KUKA KRL program: EPS_2_251806_MH13A_A_20260223023042.src

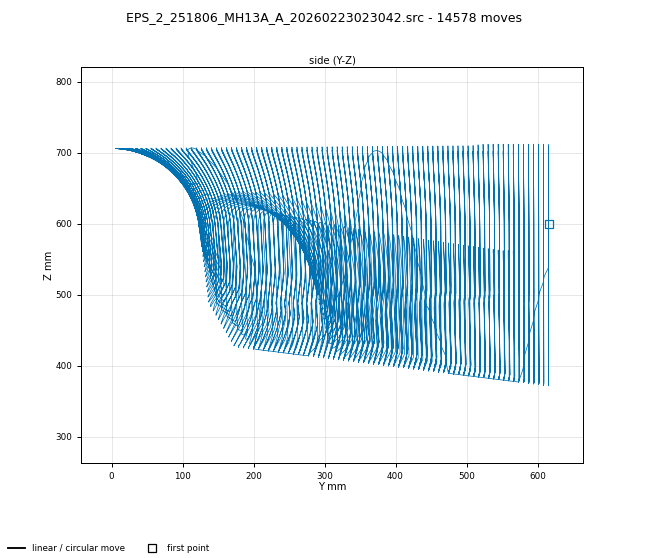
[picture p0: tool path of EPS_2_251806_MH13A_A_20260223023042.src, 14578 of 14580 moves have a stored position in this frame; points joined in program order, loops and branches not executed]
&ACCESS RVP
&REL 4
&COMMENT QRS 19112012
&PARAM EDITMASK = *
DEF PART()
EXT BAS (BAS_COMMAND :IN,REAL :IN )
INT I
BAS (#INITMOV,0 )

;KUKA QRS Post kuka4.cps  Date:22-06-2017 !

File_ID=3082

QRS_PRE_INIT()

;Init var - Until changes are made in qrs_pre_init
Outlet_Square_prg=0
Inlet_1_Square_prg=0
Inlet_2_Square_prg=0
Inlet_3_Square_prg=0
Inlet_4_Square_prg=0
Inlet_5_Square_prg=0

Outlet_1={X 0.000, Y 524.580, Z 611.500, B 0.000, E1 0.000 }
Inlet_1={X 0.000, Y 548.820, Z 271.500, B 0.000, E1 90.000 }
Inlet_2={X 0.000, Y 525.290, Z 601.500, B 0.000, E1 180.000 }
Outlet_1_type=201
Inlet_1_type=201
Inlet_2_type=201
;QRS#1=Sidecore dimensions
;QRS#2=200-8" PVC SDR 35
;QRS#3=200-8" PVC SDR 35
;QRS#4=200-8" PVC SDR 35
;QRS#5=
;QRS#6=
;QRS#7=
;QRS#8=
;QRS#9=12-08 PSX
;QRS#10=12-08 PSX
;QRS#11=12-08 PSX
;QRS#12=
;QRS#13=
;QRS#14=
;QRS#15=
;QRS#16=1220x127x991 3,25'
;QRS#17=EPS Height
;QRS#18=712
;QRS#19=*
;QRS#20= UPDATED VERSION 22-06-2017
;QRS#21=*
Outlet_Square=0100
Inlet_1_Square=0100
Inlet_2_Square=0100
Inlet_3_Square=0
Inlet_4_Square=0
Inlet_5_Square=0
Mill_Square=1
Outlet_Square_Prg=204
Inlet_1_Square_prg=204
Inlet_2_Square_prg=204

QRS_INIT()

$ADVANCE=5

; T1
PTP {E1 173.498,E2 173.498}
PTP {X 0,Y 615.498,A -85,B 0,C 180,E1 173.498,E2 173.498,E3 0,E4 0,E5 0,E6 0}
QRS_SPEED_INIT()
LIN {X 0,Y 615.498,Z 600,A -85,B 0,C 180,E1 173.498,E2 173.498,E3 0,E4 0,E5 0,E6 0} C_VEL
LIN {X 0,Y 615.498,Z 552.731,A -85,B 0,C 180,E1 173.498,E2 173.498} C_VEL
LIN {X 0,Y 615.498,Z 541.852,A -85,B 0,C 180,E1 173.498,E2 173.498} C_VEL
LIN {X 0,Y 615.496,Z 540.208,A -85,B 0,C 180,E1 173.418,E2 173.418} C_VEL
LIN {X 0,Y 615.497,Z 532.536,A -85,B 0,C 180,E1 172.455,E2 172.455} C_VEL
LIN {X 0,Y 615.498,Z 522.758,A -85,B 0,C 180,E1 171.463,E2 171.463} C_VEL
LIN {X 0,Y 615.498,Z 512.492,A -85,B 0,C 180,E1 170.636,E2 170.636} C_VEL
LIN {X 0,Y 615.496,Z 500.928,A -85,B 0,C 180,E1 169.889,E2 169.889} C_VEL
LIN {X 0,Y 615.499,Z 489.021,A -85,B 0,C 180,E1 169.291,E2 169.291} C_VEL
LIN {X 0,Y 615.498,Z 476.155,A -85,B 0,C 180,E1 168.807,E2 168.807} C_VEL
LIN {X 0,Y 615.497,Z 463.553,A -85,B 0,C 180,E1 168.473,E2 168.473} C_VEL
LIN {X 0,Y 615.498,Z 450.425,A -85,B 0,C 180,E1 168.265,E2 168.265} C_VEL
LIN {X 0,Y 615.498,Z 372.93,A -85,B 0,C 180,E1 167.344,E2 167.344} C_VEL
LIN {X 0,Y 615.495,Z 371.855,A -85,B 0,C 180,E1 167.218,E2 167.218} C_VEL
LIN {X 0,Y 615.472,Z 371.694,A -85,B 0,C 180,E1 164.773,E2 164.773} C_VEL
LIN {X 0,Y 615.491,Z 371.682,A -85,B 0,C 180,E1 162.043,E2 162.043} C_VEL
LIN {X 0,Y 615.495,Z 371.698,A -85,B 0,C 180,E1 159.269,E2 159.269} C_VEL
LIN {X 0,Y 615.469,Z 371.687,A -85,B 0,C 180,E1 156.443,E2 156.443} C_VEL
LIN {X 0,Y 615.487,Z 371.692,A -85,B 0,C 180,E1 153.556,E2 153.556} C_VEL
LIN {X 0,Y 615.491,Z 371.699,A -85,B 0,C 180,E1 151.342,E2 151.342} C_VEL
LIN {X 0,Y 615.47,Z 371.695,A -85,B 0,C 180,E1 148.917,E2 148.917} C_VEL
LIN {X 0,Y 615.464,Z 371.688,A -85,B 0,C 180,E1 146.47,E2 146.47} C_VEL
LIN {X 0,Y 615.483,Z 371.684,A -85,B 0,C 180,E1 144.167,E2 144.167} C_VEL
LIN {X 0,Y 615.475,Z 371.697,A -85,B 0,C 180,E1 141.094,E2 141.094} C_VEL
LIN {X 0,Y 615.46,Z 371.689,A -85,B 0,C 180,E1 138.524,E2 138.524} C_VEL
LIN {X 0,Y 615.493,Z 371.686,A -85,B 0,C 180,E1 135.851,E2 135.851} C_VEL
LIN {X 0,Y 615.467,Z 371.696,A -85,B 0,C 180,E1 133.045,E2 133.045} C_VEL
LIN {X 0,Y 615.455,Z 371.69,A -85,B 0,C 180,E1 130.609,E2 130.609} C_VEL
LIN {X 0,Y 615.482,Z 371.687,A -85,B 0,C 180,E1 128.011,E2 128.011} C_VEL
LIN {X 0,Y 615.494,Z 371.695,A -85,B 0,C 180,E1 125.616,E2 125.616} C_VEL
LIN {X 0,Y 615.474,Z 371.698,A -85,B 0,C 180,E1 123.237,E2 123.237} C_VEL
LIN {X 0,Y 615.452,Z 371.694,A -85,B 0,C 180,E1 120.922,E2 120.922} C_VEL
LIN {X 0,Y 615.457,Z 371.689,A -85,B 0,C 180,E1 118.444,E2 118.444} C_VEL
LIN {X 0,Y 615.494,Z 371.701,A -85,B 0,C 180,E1 115.569,E2 115.569} C_VEL
LIN {X 0,Y 615.498,Z 372.248,A -85,B 0,C 180,E1 115.334,E2 115.334} C_VEL
LIN {X 0,Y 615.455,Z 395.722,A -85,B 0,C 180,E1 112.721,E2 112.721} C_VEL
LIN {X 0,Y 615.489,Z 421.96,A -85,B 0,C 180,E1 109.859,E2 109.859} C_VEL
LIN {X 0,Y 615.449,Z 447.71,A -85,B 0,C 180,E1 107.1,E2 107.1} C_VEL
LIN {X 0,Y 615.495,Z 473.284,A -85,B 0,C 180,E1 104.395,E2 104.395} C_VEL
LIN {X 0,Y 615.494,Z 488.065,A -85,B 0,C 180,E1 102.865,E2 102.865} C_VEL
LIN {X 0,Y 615.482,Z 504.142,A -85,B 0,C 180,E1 102.656,E2 102.656} C_VEL
LIN {X 0,Y 615.493,Z 597.644,A -85,B 0,C 180,E1 101.547,E2 101.547} C_VEL
LIN {X 0,Y 615.499,Z 610.222,A -85,B 0,C 180,E1 101.276,E2 101.276} C_VEL
LIN {X 0,Y 615.497,Z 623.523,A -85,B 0,C 180,E1 100.845,E2 100.845} C_VEL
LIN {X 0,Y 615.493,Z 634.565,A -85,B 0,C 180,E1 100.36,E2 100.36} C_VEL
LIN {X 0,Y 615.491,Z 646.305,A -85,B 0,C 180,E1 99.696,E2 99.696} C_VEL
LIN {X 0,Y 615.499,Z 656.768,A -85,B 0,C 180,E1 98.95,E2 98.95} C_VEL
LIN {X 0,Y 615.498,Z 665.331,A -85,B 0,C 180,E1 98.206,E2 98.206} C_VEL
LIN {X 0,Y 615.497,Z 673.21,A -85,B 0,C 180,E1 97.38,E2 97.38} C_VEL
LIN {X 0,Y 615.497,Z 680.899,A -85,B 0,C 180,E1 96.392,E2 96.392} C_VEL
LIN {X 0,Y 615.497,Z 687.958,A -85,B 0,C 180,E1 95.241,E2 95.241} C_VEL
LIN {X 0,Y 615.494,Z 692.658,A -85,B 0,C 180,E1 94.256,E2 94.256} C_VEL
LIN {X 0,Y 615.494,Z 696.255,A -85,B 0,C 180,E1 93.273,E2 93.273} C_VEL
LIN {X 0,Y 615.496,Z 698.115,A -85,B 0,C 180,E1 92.618,E2 92.618} C_VEL
LIN {X 0,Y 615.499,Z 699.533,A -85,B 0,C 180,E1 91.963,E2 91.963} C_VEL
LIN {X 0,Y 615.496,Z 701.142,A -85,B 0,C 180,E1 90.654,E2 90.654} C_VEL
LIN {X 0,Y 615.495,Z 701.384,A -85,B 0,C 180,E1 90,E2 90} C_VEL
LIN {X 0,Y 615.495,Z 701.206,A -85,B 0,C 180,E1 89.346,E2 89.346} C_VEL
LIN {X 0,Y 615.499,Z 699.682,A -85,B 0,C 180,E1 88.037,E2 88.037} C_VEL
LIN {X 0,Y 615.498,Z 698.341,A -85,B 0,C 180,E1 87.382,E2 87.382} C_VEL
LIN {X 0,Y 615.496,Z 695.494,A -85,B 0,C 180,E1 86.399,E2 86.399} C_VEL
LIN {X 0,Y 615.498,Z 691.634,A -85,B 0,C 180,E1 85.415,E2 85.415} C_VEL
LIN {X 0,Y 615.498,Z 686.651,A -85,B 0,C 180,E1 84.43,E2 84.43} C_VEL
LIN {X 0,Y 615.496,Z 680.208,A -85,B 0,C 180,E1 83.418,E2 83.418} C_VEL
LIN {X 0,Y 615.497,Z 672.535,A -85,B 0,C 180,E1 82.454,E2 82.454} C_VEL
LIN {X 0,Y 615.498,Z 662.757,A -85,B 0,C 180,E1 81.463,E2 81.463} C_VEL
LIN {X 0,Y 615.498,Z 652.491,A -85,B 0,C 180,E1 80.635,E2 80.635} C_VEL
LIN {X 0,Y 615.492,Z 640.927,A -85,B 0,C 180,E1 79.889,E2 79.889} C_VEL
LIN {X 0,Y 615.497,Z 629.02,A -85,B 0,C 180,E1 79.291,E2 79.291} C_VEL
LIN {X 0,Y 615.498,Z 616.153,A -85,B 0,C 180,E1 78.807,E2 78.807} C_VEL
LIN {X 0,Y 615.493,Z 603.55,A -85,B 0,C 180,E1 78.473,E2 78.473} C_VEL
LIN {X 0,Y 615.491,Z 590.42,A -85,B 0,C 180,E1 78.264,E2 78.264} C_VEL
LIN {X 0,Y 615.489,Z 488.172,A -85,B 0,C 180,E1 77.05,E2 77.05} C_VEL
LIN {X 0,Y 615.453,Z 466.245,A -85,B 0,C 180,E1 74.773,E2 74.773} C_VEL
LIN {X 0,Y 615.495,Z 440.506,A -85,B 0,C 180,E1 72.043,E2 72.043} C_VEL
LIN {X 0,Y 615.494,Z 414.735,A -85,B 0,C 180,E1 69.269,E2 69.269} C_VEL
LIN {X 0,Y 615.448,Z 390.567,A -85,B 0,C 180,E1 66.62,E2 66.62} C_VEL
LIN {X 0,Y 615.497,Z 372.017,A -85,B 0,C 180,E1 64.539,E2 64.539} C_VEL
LIN {X 0,Y 615.497,Z 371.697,A -85,B 0,C 180,E1 64.284,E2 64.284} C_VEL
LIN {X 0,Y 615.441,Z 371.692,A -85,B 0,C 180,E1 61.339,E2 61.339} C_VEL
LIN {X 0,Y 615.445,Z 371.696,A -85,B 0,C 180,E1 58.921,E2 58.921} C_VEL
LIN {X 0,Y 615.492,Z 371.689,A -85,B 0,C 180,E1 55.978,E2 55.978} C_VEL
LIN {X 0,Y 615.451,Z 371.691,A -85,B 0,C 180,E1 53.572,E2 53.572} C_VEL
LIN {X 0,Y 615.442,Z 371.696,A -85,B 0,C 180,E1 50.944,E2 50.944} C_VEL
LIN {X 0,Y 615.471,Z 371.7,A -85,B 0,C 180,E1 48.524,E2 48.524} C_VEL
LIN {X 0,Y 615.479,Z 371.689,A -85,B 0,C 180,E1 45.849,E2 45.849} C_VEL
LIN {X 0,Y 615.436,Z 371.693,A -85,B 0,C 180,E1 43.249,E2 43.249} C_VEL
LIN {X 0,Y 615.436,Z 371.695,A -85,B 0,C 180,E1 41.088,E2 41.088} C_VEL
LIN {X 0,Y 615.441,Z 371.696,A -85,B 0,C 180,E1 38.908,E2 38.908} C_VEL
LIN {X 0,Y 615.479,Z 371.701,A -85,B 0,C 180,E1 36.426,E2 36.426} C_VEL
LIN {X 0,Y 615.447,Z 371.692,A -85,B 0,C 180,E1 33.528,E2 33.528} C_VEL
LIN {X 0,Y 615.434,Z 371.695,A -85,B 0,C 180,E1 31.077,E2 31.077} C_VEL
LIN {X 0,Y 615.479,Z 371.699,A -85,B 0,C 180,E1 28.448,E2 28.448} C_VEL
LIN {X 0,Y 615.448,Z 371.692,A -85,B 0,C 180,E1 25.56,E2 25.56} C_VEL
LIN {X 0,Y 615.448,Z 371.692,A -85,B 0,C 180,E1 23.558,E2 23.558} C_VEL
LIN {X 0,Y 615.439,Z 371.693,A -85,B 0,C 180,E1 21.434,E2 21.434} C_VEL
LIN {X 0,Y 615.435,Z 371.694,A -85,B 0,C 180,E1 19.34,E2 19.34} C_VEL
LIN {X 0,Y 615.431,Z 371.694,A -85,B 0,C 180,E1 17.272,E2 17.272} C_VEL
LIN {X 0,Y 615.431,Z 371.695,A -85,B 0,C 180,E1 15.228,E2 15.228} C_VEL
LIN {X 0,Y 615.43,Z 371.695,A -85,B 0,C 180,E1 13.203,E2 13.203} C_VEL
LIN {X 0,Y 615.436,Z 371.697,A -85,B 0,C 180,E1 10.861,E2 10.861} C_VEL
LIN {X 0,Y 615.461,Z 371.698,A -85,B 0,C 180,E1 8.537,E2 8.537} C_VEL
LIN {X 0,Y 615.484,Z 371.692,A -85,B 0,C 180,E1 5.899,E2 5.899} C_VEL
LIN {X 0,Y 615.43,Z 371.695,A -85,B 0,C 180,E1 3.273,E2 3.273} C_VEL
LIN {X 0,Y 615.431,Z 371.695,A -85,B 0,C 180,E1 1.309,E2 1.309} C_VEL
LIN {X 0,Y 615.432,Z 371.695,A -85,B 0,C 180,E1 -0.654,E2 -0.654} C_VEL
LIN {X 0,Y 615.433,Z 371.694,A -85,B 0,C 180,E1 -2.618,E2 -2.618} C_VEL
LIN {X 0,Y 615.435,Z 371.694,A -85,B 0,C 180,E1 -4.585,E2 -4.585} C_VEL
LIN {X 0,Y 615.436,Z 371.694,A -85,B 0,C 180,E1 -6.557,E2 -6.557} C_VEL
LIN {X 0,Y 615.437,Z 371.694,A -85,B 0,C 180,E1 -8.537,E2 -8.537} C_VEL
LIN {X 0,Y 615.425,Z 371.696,A -85,B 0,C 180,E1 -10.855,E2 -10.855} C_VEL
LIN {X 0,Y 615.433,Z 371.697,A -85,B 0,C 180,E1 -13.202,E2 -13.202} C_VEL
LIN {X 0,Y 615.49,Z 371.699,A -85,B 0,C 180,E1 -15.905,E2 -15.905} C_VEL
LIN {X 0,Y 615.429,Z 371.696,A -85,B 0,C 180,E1 -18.648,E2 -18.648} C_VEL
LIN {X 0,Y 615.426,Z 371.696,A -85,B 0,C 180,E1 -20.733,E2 -20.733} C_VEL
LIN {X 0,Y 615.423,Z 371.696,A -85,B 0,C 180,E1 -22.847,E2 -22.847} C_VEL
LIN {X 0,Y 615.423,Z 371.697,A -85,B 0,C 180,E1 -24.995,E2 -24.995} C_VEL
LIN {X 0,Y 615.483,Z 371.701,A -85,B 0,C 180,E1 -27.915,E2 -27.915} C_VEL
LIN {X 0,Y 615.475,Z 371.694,A -85,B 0,C 180,E1 -30.161,E2 -30.161} C_VEL
LIN {X 0,Y 615.441,Z 371.695,A -85,B 0,C 180,E1 -32.46,E2 -32.46} C_VEL
LIN {X 0,Y 615.421,Z 371.697,A -85,B 0,C 180,E1 -34.819,E2 -34.819} C_VEL
LIN {X 0,Y 615.429,Z 371.698,A -85,B 0,C 180,E1 -37.246,E2 -37.246} C_VEL
LIN {X 0,Y 615.486,Z 371.695,A -85,B 0,C 180,E1 -40.088,E2 -40.088} C_VEL
LIN {X 0,Y 615.45,Z 371.696,A -85,B 0,C 180,E1 -42.356,E2 -42.356} C_VEL
LIN {X 0,Y 615.417,Z 371.698,A -85,B 0,C 180,E1 -44.924,E2 -44.924} C_VEL
LIN {X 0,Y 615.417,Z 371.698,A -85,B 0,C 180,E1 -46.96,E2 -46.96} C_VEL
LIN {X 0,Y 615.417,Z 371.698,A -85,B 0,C 180,E1 -48.913,E2 -48.913} C_VEL
LIN {X 0,Y 615.419,Z 371.698,A -85,B 0,C 180,E1 -51.09,E2 -51.09} C_VEL
LIN {X 0,Y 615.453,Z 371.699,A -85,B 0,C 180,E1 -53.572,E2 -53.572} C_VEL
LIN {X 0,Y 615.437,Z 371.697,A -85,B 0,C 180,E1 -56.473,E2 -56.473} C_VEL
LIN {X 0,Y 615.415,Z 371.699,A -85,B 0,C 180,E1 -59.076,E2 -59.076} C_VEL
LIN {X 0,Y 615.448,Z 371.699,A -85,B 0,C 180,E1 -61.557,E2 -61.557} C_VEL
LIN {X 0,Y 615.498,Z 371.811,A -85,B 0,C 180,E1 -64.012,E2 -64.012} C_VEL
LIN {X 0,Y 615.497,Z 372.154,A -85,B 0,C 180,E1 -64.103,E2 -64.103} C_VEL
LIN {X 0,Y 615.463,Z 395.618,A -85,B 0,C 180,E1 -66.621,E2 -66.621} C_VEL
LIN {X 0,Y 615.473,Z 420.833,A -85,B 0,C 180,E1 -69.269,E2 -69.269} C_VEL
LIN {X 0,Y 615.496,Z 447.725,A -85,B 0,C 180,E1 -72.043,E2 -72.043} C_VEL
LIN {X 0,Y 615.456,Z 474.585,A -85,B 0,C 180,E1 -74.773,E2 -74.773} C_VEL
LIN {X 0,Y 615.491,Z 497.862,A -85,B 0,C 180,E1 -77.092,E2 -77.092} C_VEL
LIN {X 0,Y 615.492,Z 607.82,A -85,B 0,C 180,E1 -78.411,E2 -78.411} C_VEL
LIN {X 0,Y 615.499,Z 620.336,A -85,B 0,C 180,E1 -78.682,E2 -78.682} C_VEL
LIN {X 0,Y 615.496,Z 633.5,A -85,B 0,C 180,E1 -79.109,E2 -79.109} C_VEL
LIN {X 0,Y 615.491,Z 645.473,A -85,B 0,C 180,E1 -79.639,E2 -79.639} C_VEL
LIN {X 0,Y 615.492,Z 656.992,A -85,B 0,C 180,E1 -80.304,E2 -80.304} C_VEL
LIN {X 0,Y 615.499,Z 667.339,A -85,B 0,C 180,E1 -81.05,E2 -81.05} C_VEL
LIN {X 0,Y 615.497,Z 675.81,A -85,B 0,C 180,E1 -81.794,E2 -81.794} C_VEL
LIN {X 0,Y 615.498,Z 683.605,A -85,B 0,C 180,E1 -82.619,E2 -82.619} C_VEL
LIN {X 0,Y 615.496,Z 691.202,A -85,B 0,C 180,E1 -83.608,E2 -83.608} C_VEL
LIN {X 0,Y 615.498,Z 698.204,A -85,B 0,C 180,E1 -84.759,E2 -84.759} C_VEL
LIN {X 0,Y 615.494,Z 702.851,A -85,B 0,C 180,E1 -85.743,E2 -85.743} C_VEL
LIN {X 0,Y 615.494,Z 706.398,A -85,B 0,C 180,E1 -86.727,E2 -86.727} C_VEL
LIN {X 0,Y 615.497,Z 708.233,A -85,B 0,C 180,E1 -87.382,E2 -87.382} C_VEL
LIN {X 0,Y 615.499,Z 709.607,A -85,B 0,C 180,E1 -88.037,E2 -88.037} C_VEL
LIN {X 0,Y 615.496,Z 711.173,A -85,B 0,C 180,E1 -89.346,E2 -89.346} C_VEL
LIN {X 0,Y 615.494,Z 711.389,A -85,B 0,C 180,E1 -90,E2 -90} C_VEL
LIN {X 0,Y 615.495,Z 710.58,A -85,B 0,C 180,E1 -91.308,E2 -91.308} C_VEL
LIN {X 0,Y 615.499,Z 709.608,A -85,B 0,C 180,E1 -91.963,E2 -91.963} C_VEL
LIN {X 0,Y 615.497,Z 708.233,A -85,B 0,C 180,E1 -92.618,E2 -92.618} C_VEL
LIN {X 0,Y 615.496,Z 705.35,A -85,B 0,C 180,E1 -93.601,E2 -93.601} C_VEL
LIN {X 0,Y 615.498,Z 701.442,A -85,B 0,C 180,E1 -94.584,E2 -94.584} C_VEL
LIN {X 0,Y 615.499,Z 696.405,A -85,B 0,C 180,E1 -95.57,E2 -95.57} C_VEL
LIN {X 0,Y 615.497,Z 689.869,A -85,B 0,C 180,E1 -96.583,E2 -96.583} C_VEL
LIN {X 0,Y 615.497,Z 682.133,A -85,B 0,C 180,E1 -97.545,E2 -97.545} C_VEL
LIN {X 0,Y 615.498,Z 674.045,A -85,B 0,C 180,E1 -98.371,E2 -98.371} C_VEL
LIN {X 0,Y 615.499,Z 664.168,A -85,B 0,C 180,E1 -99.199,E2 -99.199} C_VEL
LIN {X 0,Y 615.492,Z 652.981,A -85,B 0,C 180,E1 -99.945,E2 -99.945} C_VEL
LIN {X 0,Y 615.493,Z 642.022,A -85,B 0,C 180,E1 -100.527,E2 -100.527} C_VEL
LIN {X 0,Y 615.499,Z 629.416,A -85,B 0,C 180,E1 -101.042,E2 -101.042} C_VEL
LIN {X 0,Y 615.498,Z 617.063,A -85,B 0,C 180,E1 -101.401,E2 -101.401} C_VEL
LIN {X 0,Y 615.491,Z 603.466,A -85,B 0,C 180,E1 -101.652,E2 -101.652} C_VEL
LIN {X 0,Y 615.491,Z 497.865,A -85,B 0,C 180,E1 -102.907,E2 -102.907} C_VEL
LIN {X 0,Y 615.456,Z 474.586,A -85,B 0,C 180,E1 -105.227,E2 -105.227} C_VEL
LIN {X 0,Y 615.496,Z 447.727,A -85,B 0,C 180,E1 -107.957,E2 -107.957} C_VEL
LIN {X 0,Y 615.473,Z 420.835,A -85,B 0,C 180,E1 -110.731,E2 -110.731} C_VEL
LIN {X 0,Y 615.463,Z 395.62,A -85,B 0,C 180,E1 -113.379,E2 -113.379} C_VEL
LIN {X 0,Y 615.495,Z 372.155,A -85,B 0,C 180,E1 -115.897,E2 -115.897} C_VEL
LIN {X 0,Y 615.496,Z 371.721,A -85,B 0,C 180,E1 -116.079,E2 -116.079} C_VEL
LIN {X 0,Y 615.423,Z 371.7,A -85,B 0,C 180,E1 -118.661,E2 -118.661} C_VEL
LIN {X 0,Y 615.411,Z 371.7,A -85,B 0,C 180,E1 -121.074,E2 -121.074} C_VEL
LIN {X 0,Y 615.441,Z 371.7,A -85,B 0,C 180,E1 -123.527,E2 -123.527} C_VEL
LIN {X 0,Y 615.443,Z 371.697,A -85,B 0,C 180,E1 -126.428,E2 -126.428} C_VEL
LIN {X 0,Y 615.421,Z 371.698,A -85,B 0,C 180,E1 -128.91,E2 -128.91} C_VEL
LIN {X 0,Y 615.427,Z 371.698,A -85,B 0,C 180,E1 -131.088,E2 -131.088} C_VEL
LIN {X 0,Y 615.438,Z 371.698,A -85,B 0,C 180,E1 -133.249,E2 -133.249} C_VEL
LIN {X 0,Y 615.486,Z 371.694,A -85,B 0,C 180,E1 -136.003,E2 -136.003} C_VEL
LIN {X 0,Y 615.444,Z 371.693,A -85,B 0,C 180,E1 -138.522,E2 -138.522} C_VEL
LIN {X 0,Y 615.438,Z 371.695,A -85,B 0,C 180,E1 -140.944,E2 -140.944} C_VEL
LIN {X 0,Y 615.482,Z 371.702,A -85,B 0,C 180,E1 -143.575,E2 -143.575} C_VEL
LIN {X 0,Y 615.453,Z 371.691,A -85,B 0,C 180,E1 -146.471,E2 -146.471} C_VEL
LIN {X 0,Y 615.456,Z 371.696,A -85,B 0,C 180,E1 -149.078,E2 -149.078} C_VEL
LIN {X 0,Y 615.494,Z 371.699,A -85,B 0,C 180,E1 -151.549,E2 -151.549} C_VEL
LIN {X 0,Y 615.46,Z 371.689,A -85,B 0,C 180,E1 -154.437,E2 -154.437} C_VEL
LIN {X 0,Y 615.474,Z 371.698,A -85,B 0,C 180,E1 -157.155,E2 -157.155} C_VEL
LIN {X 0,Y 615.487,Z 371.686,A -85,B 0,C 180,E1 -159.967,E2 -159.967} C_VEL
LIN {X 0,Y 615.462,Z 371.692,A -85,B 0,C 180,E1 -162.729,E2 -162.729} C_VEL
LIN {X 0,Y 615.486,Z 371.696,A -85,B 0,C 180,E1 -165.451,E2 -165.451} C_VEL
LIN {X 0,Y 615.496,Z 371.905,A -85,B 0,C 180,E1 -167.323,E2 -167.323} C_VEL
LIN {X 0,Y 615.497,Z 372.808,A -85,B 0,C 180,E1 -167.428,E2 -167.428} C_VEL
LIN {X 0,Y 615.497,Z 458.789,A -85,B 0,C 180,E1 -168.473,E2 -168.473} C_VEL
LIN {X 0,Y 615.498,Z 471.737,A -85,B 0,C 180,E1 -168.765,E2 -168.765} C_VEL
LIN {X 0,Y 615.498,Z 484.736,A -85,B 0,C 180,E1 -169.2,E2 -169.2} C_VEL
LIN {X 0,Y 615.497,Z 496.194,A -85,B 0,C 180,E1 -169.723,E2 -169.723} C_VEL
LIN {X 0,Y 615.491,Z 507.576,A -85,B 0,C 180,E1 -170.387,E2 -170.387} C_VEL
LIN {X 0,Y 615.498,Z 517.823,A -85,B 0,C 180,E1 -171.133,E2 -171.133} C_VEL
LIN {X 0,Y 615.499,Z 527.034,A -85,B 0,C 180,E1 -171.959,E2 -171.959} C_VEL
LIN {X 0,Y 615.499,Z 535.892,A -85,B 0,C 180,E1 -172.943,E2 -172.943} C_VEL
LIN {X 0,Y 615.497,Z 543.123,A -85,B 0,C 180,E1 -173.937,E2 -173.937} C_VEL
LIN {X 0,Y 615.497,Z 547.958,A -85,B 0,C 180,E1 -174.759,E2 -174.759} C_VEL
LIN {X 0,Y 615.494,Z 552.658,A -85,B 0,C 180,E1 -175.744,E2 -175.744} C_VEL
LIN {X 0,Y 615.494,Z 556.255,A -85,B 0,C 180,E1 -176.727,E2 -176.727} C_VEL
LIN {X 0,Y 615.496,Z 558.115,A -85,B 0,C 180,E1 -177.382,E2 -177.382} C_VEL
LIN {X 0,Y 615.499,Z 559.533,A -85,B 0,C 180,E1 -178.037,E2 -178.037} C_VEL
LIN {X 0,Y 615.496,Z 561.142,A -85,B 0,C 180,E1 -179.346,E2 -179.346} C_VEL
LIN {X 0,Y 615.495,Z 561.384,A -85,B 0,C 180,E1 -180,E2 -180} C_VEL
LIN {X 0,Y 615.495,Z 561.206,A -85,B 0,C 180,E1 -180.654,E2 -180.654} C_VEL
LIN {X 0,Y 615.499,Z 559.682,A -85,B 0,C 180,E1 -181.963,E2 -181.963} C_VEL
LIN {X 0,Y 615.498,Z 558.341,A -85,B 0,C 180,E1 -182.618,E2 -182.618} C_VEL
LIN {X 0,Y 615.496,Z 555.494,A -85,B 0,C 180,E1 -183.601,E2 -183.601} C_VEL
LIN {X 0,Y 615.498,Z 551.634,A -85,B 0,C 180,E1 -184.585,E2 -184.585} C_VEL
LIN {X 0,Y 615.498,Z 546.651,A -85,B 0,C 180,E1 -185.57,E2 -185.57} C_VEL
LIN {X 0,Y 615.496,Z 540.208,A -85,B 0,C 180,E1 -186.582,E2 -186.582} C_VEL
LIN {X 0,Y 614.829,Z 537.026,A -85,B 0,C 180,E1 -187.031,E2 -187.031} C_VEL
LIN {X 0,Y 611.989,Z 531.453,A -85,B 0,C 180,E1 -187.748,E2 -187.748} C_VEL
LIN {X 0,Y 609.138,Z 525.177,A -85,B 0,C 180,E1 -188.429,E2 -188.429} C_VEL
LIN {X 0,Y 608.477,Z 520.936,A -85,B 0,C 180,E1 -188.819,E2 -188.819} C_VEL
LIN {X 0,Y 608.496,Z 510.391,A -85,B 0,C 180,E1 -189.641,E2 -189.641} C_VEL
LIN {X 0,Y 608.497,Z 499.604,A -85,B 0,C 180,E1 -190.313,E2 -190.313} C_VEL
LIN {X 0,Y 608.537,Z 487.826,A -85,B 0,C 180,E1 -190.889,E2 -190.889} C_VEL
LIN {X 0,Y 608.534,Z 476.24,A -85,B 0,C 180,E1 -191.323,E2 -191.323} C_VEL
LIN {X 0,Y 608.548,Z 463.627,A -85,B 0,C 180,E1 -191.66,E2 -191.66} C_VEL
LIN {X 0,Y 608.551,Z 450.534,A -85,B 0,C 180,E1 -191.871,E2 -191.871} C_VEL
LIN {X 0,Y 608.606,Z 374.059,A -85,B 0,C 180,E1 -192.78,E2 -192.78} C_VEL
LIN {X 0,Y 608.506,Z 372.86,A -85,B 0,C 180,E1 -192.888,E2 -192.888} C_VEL
LIN {X 0,Y 608.462,Z 372.688,A -85,B 0,C 180,E1 -195.406,E2 -195.406} C_VEL
LIN {X 0,Y 608.451,Z 372.689,A -85,B 0,C 180,E1 -198.172,E2 -198.172} C_VEL
LIN {X 0,Y 608.456,Z 372.695,A -85,B 0,C 180,E1 -200.982,E2 -200.982} C_VEL
LIN {X 0,Y 608.446,Z 372.693,A -85,B 0,C 180,E1 -203.124,E2 -203.124} C_VEL
LIN {X 0,Y 608.459,Z 372.686,A -85,B 0,C 180,E1 -205.718,E2 -205.718} C_VEL
LIN {X 0,Y 608.476,Z 372.693,A -85,B 0,C 180,E1 -208.62,E2 -208.62} C_VEL
LIN {X 0,Y 608.443,Z 372.69,A -85,B 0,C 180,E1 -211.318,E2 -211.318} C_VEL
LIN {X 0,Y 608.449,Z 372.687,A -85,B 0,C 180,E1 -213.731,E2 -213.731} C_VEL
LIN {X 0,Y 608.449,Z 372.689,A -85,B 0,C 180,E1 -216.092,E2 -216.092} C_VEL
LIN {X 0,Y 608.464,Z 372.695,A -85,B 0,C 180,E1 -218.589,E2 -218.589} C_VEL
LIN {X 0,Y 608.44,Z 372.69,A -85,B 0,C 180,E1 -221.34,E2 -221.34} C_VEL
LIN {X 0,Y 608.46,Z 372.691,A -85,B 0,C 180,E1 -224.264,E2 -224.264} C_VEL
LIN {X 0,Y 608.433,Z 372.693,A -85,B 0,C 180,E1 -227.038,E2 -227.038} C_VEL
LIN {X 0,Y 608.456,Z 372.687,A -85,B 0,C 180,E1 -229.697,E2 -229.697} C_VEL
LIN {X 0,Y 608.465,Z 372.691,A -85,B 0,C 180,E1 -232.253,E2 -232.253} C_VEL
LIN {X 0,Y 608.423,Z 372.693,A -85,B 0,C 180,E1 -235.099,E2 -235.099} C_VEL
LIN {X 0,Y 608.438,Z 372.689,A -85,B 0,C 180,E1 -237.482,E2 -237.482} C_VEL
LIN {X 0,Y 608.478,Z 372.69,A -85,B 0,C 180,E1 -240.221,E2 -240.221} C_VEL
LIN {X 0,Y 608.419,Z 372.694,A -85,B 0,C 180,E1 -243.224,E2 -243.224} C_VEL
LIN {X 0,Y 608.512,Z 372.852,A -85,B 0,C 180,E1 -244.409,E2 -244.409} C_VEL
LIN {X 0,Y 608.72,Z 376.879,A -85,B 0,C 180,E1 -244.894,E2 -244.894} C_VEL
LIN {X 0,Y 608.638,Z 404.252,A -85,B 0,C 180,E1 -247.958,E2 -247.958} C_VEL
LIN {X 0,Y 608.587,Z 430.016,A -85,B 0,C 180,E1 -250.785,E2 -250.785} C_VEL
LIN {X 0,Y 608.504,Z 456.571,A -85,B 0,C 180,E1 -253.647,E2 -253.647} C_VEL
LIN {X 0,Y 608.5,Z 481.548,A -85,B 0,C 180,E1 -256.304,E2 -256.304} C_VEL
LIN {X 0,Y 608.525,Z 488.12,A -85,B 0,C 180,E1 -256.985,E2 -256.985} C_VEL
LIN {X 0,Y 608.572,Z 497.08,A -85,B 0,C 180,E1 -257.113,E2 -257.113} C_VEL
LIN {X 0,Y 608.551,Z 597.792,A -85,B 0,C 180,E1 -258.319,E2 -258.319} C_VEL
LIN {X 0,Y 608.539,Z 611.104,A -85,B 0,C 180,E1 -258.614,E2 -258.614} C_VEL
LIN {X 0,Y 608.529,Z 624.346,A -85,B 0,C 180,E1 -259.055,E2 -259.055} C_VEL
LIN {X 0,Y 608.503,Z 636.366,A -85,B 0,C 180,E1 -259.603,E2 -259.603} C_VEL
LIN {X 0,Y 608.504,Z 647.786,A -85,B 0,C 180,E1 -260.275,E2 -260.275} C_VEL
LIN {X 0,Y 608.474,Z 658.079,A -85,B 0,C 180,E1 -261.029,E2 -261.029} C_VEL
LIN {X 0,Y 608.464,Z 667.352,A -85,B 0,C 180,E1 -261.866,E2 -261.866} C_VEL
LIN {X 0,Y 608.466,Z 676.325,A -85,B 0,C 180,E1 -262.867,E2 -262.867} C_VEL
LIN {X 0,Y 608.444,Z 683.555,A -85,B 0,C 180,E1 -263.867,E2 -263.867} C_VEL
LIN {X 0,Y 608.462,Z 688.434,A -85,B 0,C 180,E1 -264.698,E2 -264.698} C_VEL
LIN {X 0,Y 608.439,Z 693.178,A -85,B 0,C 180,E1 -265.694,E2 -265.694} C_VEL
LIN {X 0,Y 608.425,Z 696.811,A -85,B 0,C 180,E1 -266.689,E2 -266.689} C_VEL
LIN {X 0,Y 608.425,Z 698.691,A -85,B 0,C 180,E1 -267.352,E2 -267.352} C_VEL
LIN {X 0,Y 608.444,Z 700.127,A -85,B 0,C 180,E1 -268.014,E2 -268.014} C_VEL
LIN {X 0,Y 608.439,Z 701.752,A -85,B 0,C 180,E1 -269.338,E2 -269.338} C_VEL
LIN {X 0,Y 608.435,Z 701.995,A -85,B 0,C 180,E1 -270,E2 -270} C_VEL
LIN {X 0,Y 608.438,Z 701.815,A -85,B 0,C 180,E1 -270.662,E2 -270.662} C_VEL
LIN {X 0,Y 608.444,Z 700.276,A -85,B 0,C 180,E1 -271.986,E2 -271.986} C_VEL
LIN {X 0,Y 608.426,Z 698.917,A -85,B 0,C 180,E1 -272.648,E2 -272.648} C_VEL
LIN {X 0,Y 608.449,Z 696.04,A -85,B 0,C 180,E1 -273.642,E2 -273.642} C_VEL
LIN {X 0,Y 608.433,Z 692.141,A -85,B 0,C 180,E1 -274.638,E2 -274.638} C_VEL
LIN {X 0,Y 608.449,Z 687.111,A -85,B 0,C 180,E1 -275.635,E2 -275.635} C_VEL
LIN {X 0,Y 608.441,Z 680.794,A -85,B 0,C 180,E1 -276.633,E2 -276.633} C_VEL
LIN {X 0,Y 608.475,Z 672.875,A -85,B 0,C 180,E1 -277.633,E2 -277.633} C_VEL
LIN {X 0,Y 608.472,Z 663.03,A -85,B 0,C 180,E1 -278.636,E2 -278.636} C_VEL
LIN {X 0,Y 608.48,Z 652.713,A -85,B 0,C 180,E1 -279.474,E2 -279.474} C_VEL
LIN {X 0,Y 608.489,Z 641.098,A -85,B 0,C 180,E1 -280.229,E2 -280.229} C_VEL
LIN {X 0,Y 608.529,Z 629.852,A -85,B 0,C 180,E1 -280.803,E2 -280.803} C_VEL
LIN {X 0,Y 608.538,Z 617.26,A -85,B 0,C 180,E1 -281.29,E2 -281.29} C_VEL
LIN {X 0,Y 608.542,Z 603.646,A -85,B 0,C 180,E1 -281.66,E2 -281.66} C_VEL
LIN {X 0,Y 608.548,Z 590.527,A -85,B 0,C 180,E1 -281.871,E2 -281.871} C_VEL
LIN {X 0,Y 608.553,Z 488.802,A -85,B 0,C 180,E1 -283.078,E2 -283.078} C_VEL
LIN {X 0,Y 608.497,Z 487.231,A -85,B 0,C 180,E1 -283.186,E2 -283.186} C_VEL
LIN {X 0,Y 608.528,Z 461.454,A -85,B 0,C 180,E1 -285.92,E2 -285.92} C_VEL
LIN {X 0,Y 608.556,Z 434.064,A -85,B 0,C 180,E1 -288.867,E2 -288.867} C_VEL
LIN {X 0,Y 608.601,Z 409.896,A -85,B 0,C 180,E1 -291.509,E2 -291.509} C_VEL
LIN {X 0,Y 608.687,Z 383.715,A -85,B 0,C 180,E1 -294.425,E2 -294.425} C_VEL
LIN {X 0,Y 608.531,Z 372.965,A -85,B 0,C 180,E1 -295.658,E2 -295.658} C_VEL
LIN {X 0,Y 608.436,Z 372.695,A -85,B 0,C 180,E1 -296.036,E2 -296.036} C_VEL
LIN {X 0,Y 608.44,Z 372.689,A -85,B 0,C 180,E1 -298.614,E2 -298.614} C_VEL
LIN {X 0,Y 608.427,Z 372.69,A -85,B 0,C 180,E1 -300.548,E2 -300.548} C_VEL
LIN {X 0,Y 608.43,Z 372.691,A -85,B 0,C 180,E1 -302.882,E2 -302.882} C_VEL
LIN {X 0,Y 608.432,Z 372.694,A -85,B 0,C 180,E1 -305.279,E2 -305.279} C_VEL
LIN {X 0,Y 608.459,Z 372.688,A -85,B 0,C 180,E1 -308.239,E2 -308.239} C_VEL
LIN {X 0,Y 608.418,Z 372.694,A -85,B 0,C 180,E1 -311.18,E2 -311.18} C_VEL
LIN {X 0,Y 608.466,Z 372.692,A -85,B 0,C 180,E1 -313.87,E2 -313.87} C_VEL
LIN {X 0,Y 608.432,Z 372.69,A -85,B 0,C 180,E1 -316.696,E2 -316.696} C_VEL
LIN {X 0,Y 608.407,Z 372.693,A -85,B 0,C 180,E1 -318.819,E2 -318.819} C_VEL
LIN {X 0,Y 608.415,Z 372.698,A -85,B 0,C 180,E1 -321.408,E2 -321.408} C_VEL
LIN {X 0,Y 608.447,Z 372.694,A -85,B 0,C 180,E1 -323.955,E2 -323.955} C_VEL
LIN {X 0,Y 608.447,Z 372.689,A -85,B 0,C 180,E1 -326.328,E2 -326.328} C_VEL
LIN {X 0,Y 608.431,Z 372.69,A -85,B 0,C 180,E1 -328.736,E2 -328.736} C_VEL
LIN {X 0,Y 608.43,Z 372.695,A -85,B 0,C 180,E1 -331.388,E2 -331.388} C_VEL
LIN {X 0,Y 608.449,Z 372.689,A -85,B 0,C 180,E1 -334.285,E2 -334.285} C_VEL
LIN {X 0,Y 608.459,Z 372.69,A -85,B 0,C 180,E1 -336.155,E2 -336.155} C_VEL
LIN {X 0,Y 608.446,Z 372.69,A -85,B 0,C 180,E1 -338.307,E2 -338.307} C_VEL
LIN {X 0,Y 608.434,Z 372.691,A -85,B 0,C 180,E1 -341.13,E2 -341.13} C_VEL
LIN {X 0,Y 608.455,Z 372.694,A -85,B 0,C 180,E1 -343.906,E2 -343.906} C_VEL
LIN {X 0,Y 608.423,Z 372.691,A -85,B 0,C 180,E1 -346.643,E2 -346.643} C_VEL
LIN {X 0,Y 608.433,Z 372.693,A -85,B 0,C 180,E1 -349.35,E2 -349.35} C_VEL
LIN {X 0,Y 608.47,Z 372.691,A -85,B 0,C 180,E1 -352.033,E2 -352.033} C_VEL
LIN {X 0,Y 608.417,Z 372.691,A -85,B 0,C 180,E1 -354.698,E2 -354.698} C_VEL
LIN {X 0,Y 608.445,Z 372.692,A -85,B 0,C 180,E1 -357.352,E2 -357.352} C_VEL
LIN {X 0,Y 608.477,Z 372.691,A -85,B 0,C 180,E1 -360,E2 -360} C_VEL
LIN {X 0,Y 608.43,Z 372.69,A -85,B 0,C 180,E1 -362.648,E2 -362.648} C_VEL
LIN {X 0,Y 608.426,Z 372.693,A -85,B 0,C 180,E1 -365.302,E2 -365.302} C_VEL
LIN {X 0,Y 608.476,Z 372.691,A -85,B 0,C 180,E1 -367.967,E2 -367.967} C_VEL
LIN {X 0,Y 608.415,Z 372.692,A -85,B 0,C 180,E1 -370.651,E2 -370.651} C_VEL
LIN {X 0,Y 608.404,Z 372.693,A -85,B 0,C 180,E1 -372.678,E2 -372.678} C_VEL
LIN {X 0,Y 608.4,Z 372.693,A -85,B 0,C 180,E1 -374.722,E2 -374.722} C_VEL
LIN {X 0,Y 608.41,Z 372.692,A -85,B 0,C 180,E1 -376.785,E2 -376.785} C_VEL
LIN {X 0,Y 608.424,Z 372.697,A -85,B 0,C 180,E1 -379.572,E2 -379.572} C_VEL
LIN {X 0,Y 608.434,Z 372.69,A -85,B 0,C 180,E1 -382.469,E2 -382.469} C_VEL
LIN {X 0,Y 608.419,Z 372.692,A -85,B 0,C 180,E1 -384.573,E2 -384.573} C_VEL
LIN {X 0,Y 608.395,Z 372.694,A -85,B 0,C 180,E1 -386.777,E2 -386.777} C_VEL
LIN {X 0,Y 608.477,Z 372.694,A -85,B 0,C 180,E1 -389.779,E2 -389.779} C_VEL
LIN {X 0,Y 608.424,Z 372.692,A -85,B 0,C 180,E1 -392.516,E2 -392.516} C_VEL
LIN {X 0,Y 608.391,Z 372.694,A -85,B 0,C 180,E1 -394.897,E2 -394.897} C_VEL
LIN {X 0,Y 608.423,Z 372.692,A -85,B 0,C 180,E1 -397.152,E2 -397.152} C_VEL
LIN {X 0,Y 608.42,Z 372.695,A -85,B 0,C 180,E1 -399.444,E2 -399.444} C_VEL
LIN {X 0,Y 608.424,Z 372.694,A -85,B 0,C 180,E1 -402.33,E2 -402.33} C_VEL
LIN {X 0,Y 608.4,Z 372.694,A -85,B 0,C 180,E1 -404.801,E2 -404.801} C_VEL
LIN {X 0,Y 608.39,Z 372.695,A -85,B 0,C 180,E1 -407.034,E2 -407.034} C_VEL
LIN {X 0,Y 608.39,Z 372.694,A -85,B 0,C 180,E1 -408.818,E2 -408.818} C_VEL
LIN {X 0,Y 608.403,Z 372.693,A -85,B 0,C 180,E1 -410.711,E2 -410.711} C_VEL
LIN {X 0,Y 608.389,Z 372.695,A -85,B 0,C 180,E1 -413.08,E2 -413.08} C_VEL
LIN {X 0,Y 608.432,Z 372.694,A -85,B 0,C 180,E1 -415.528,E2 -415.528} C_VEL
LIN {X 0,Y 608.444,Z 372.699,A -85,B 0,C 180,E1 -417.904,E2 -417.904} C_VEL
LIN {X 0,Y 608.453,Z 372.693,A -85,B 0,C 180,E1 -420.219,E2 -420.219} C_VEL
LIN {X 0,Y 608.4,Z 372.696,A -85,B 0,C 180,E1 -422.808,E2 -422.808} C_VEL
LIN {X 0,Y 608.511,Z 372.934,A -85,B 0,C 180,E1 -423.864,E2 -423.864} C_VEL
LIN {X 0,Y 608.724,Z 377.801,A -85,B 0,C 180,E1 -424.418,E2 -424.418} C_VEL
LIN {X 0,Y 608.655,Z 402.51,A -85,B 0,C 180,E1 -427.082,E2 -427.082} C_VEL
LIN {X 0,Y 608.603,Z 429.239,A -85,B 0,C 180,E1 -429.907,E2 -429.907} C_VEL
LIN {X 0,Y 608.522,Z 454.454,A -85,B 0,C 180,E1 -432.525,E2 -432.525} C_VEL
LIN {X 0,Y 608.514,Z 477.988,A -85,B 0,C 180,E1 -434.938,E2 -434.938} C_VEL
LIN {X 0,Y 608.531,Z 497.9,A -85,B 0,C 180,E1 -436.942,E2 -436.942} C_VEL
LIN {X 0,Y 608.544,Z 607.937,A -85,B 0,C 180,E1 -438.276,E2 -438.276} C_VEL
LIN {X 0,Y 608.547,Z 621.21,A -85,B 0,C 180,E1 -438.572,E2 -438.572} C_VEL
LIN {X 0,Y 608.544,Z 634.329,A -85,B 0,C 180,E1 -439.009,E2 -439.009} C_VEL
LIN {X 0,Y 608.511,Z 645.632,A -85,B 0,C 180,E1 -439.519,E2 -439.519} C_VEL
LIN {X 0,Y 608.483,Z 657.195,A -85,B 0,C 180,E1 -440.191,E2 -440.191} C_VEL
LIN {X 0,Y 608.485,Z 667.592,A -85,B 0,C 180,E1 -440.946,E2 -440.946} C_VEL
LIN {X 0,Y 608.475,Z 676.11,A -85,B 0,C 180,E1 -441.699,E2 -441.699} C_VEL
LIN {X 0,Y 608.471,Z 683.959,A -85,B 0,C 180,E1 -442.534,E2 -442.534} C_VEL
LIN {X 0,Y 608.461,Z 691.286,A -85,B 0,C 180,E1 -443.484,E2 -443.484} C_VEL
LIN {X 0,Y 608.45,Z 696.865,A -85,B 0,C 180,E1 -444.365,E2 -444.365} C_VEL
LIN {X 0,Y 608.432,Z 701.95,A -85,B 0,C 180,E1 -445.362,E2 -445.362} C_VEL
LIN {X 0,Y 608.449,Z 705.896,A -85,B 0,C 180,E1 -446.358,E2 -446.358} C_VEL
LIN {X 0,Y 608.425,Z 708.809,A -85,B 0,C 180,E1 -447.352,E2 -447.352} C_VEL
LIN {X 0,Y 608.444,Z 710.201,A -85,B 0,C 180,E1 -448.014,E2 -448.014} C_VEL
LIN {X 0,Y 608.438,Z 711.783,A -85,B 0,C 180,E1 -449.338,E2 -449.338} C_VEL
LIN {X 0,Y 608.434,Z 712,A -85,B 0,C 180,E1 -450,E2 -450} C_VEL
LIN {X 0,Y 608.448,Z 711.184,A -85,B 0,C 180,E1 -451.324,E2 -451.324} C_VEL
LIN {X 0,Y 608.444,Z 710.202,A -85,B 0,C 180,E1 -451.986,E2 -451.986} C_VEL
LIN {X 0,Y 608.425,Z 708.809,A -85,B 0,C 180,E1 -452.648,E2 -452.648} C_VEL
LIN {X 0,Y 608.449,Z 705.896,A -85,B 0,C 180,E1 -453.642,E2 -453.642} C_VEL
LIN {X 0,Y 608.432,Z 701.95,A -85,B 0,C 180,E1 -454.638,E2 -454.638} C_VEL
LIN {X 0,Y 608.437,Z 695.877,A -85,B 0,C 180,E1 -455.801,E2 -455.801} C_VEL
LIN {X 0,Y 608.462,Z 689.235,A -85,B 0,C 180,E1 -456.799,E2 -456.799} C_VEL
LIN {X 0,Y 608.456,Z 680.989,A -85,B 0,C 180,E1 -457.8,E2 -457.8} C_VEL
LIN {X 0,Y 608.472,Z 672.536,A -85,B 0,C 180,E1 -458.636,E2 -458.636} C_VEL
LIN {X 0,Y 608.478,Z 662.091,A -85,B 0,C 180,E1 -459.473,E2 -459.473} C_VEL
LIN {X 0,Y 608.502,Z 651.756,A -85,B 0,C 180,E1 -460.145,E2 -460.145} C_VEL
LIN {X 0,Y 608.523,Z 640.24,A -85,B 0,C 180,E1 -460.741,E2 -460.741} C_VEL
LIN {X 0,Y 608.533,Z 628.874,A -85,B 0,C 180,E1 -461.193,E2 -461.193} C_VEL
LIN {X 0,Y 608.558,Z 615.353,A -85,B 0,C 180,E1 -461.575,E2 -461.575} C_VEL
LIN {X 0,Y 608.552,Z 602.085,A -85,B 0,C 180,E1 -461.808,E2 -461.808} C_VEL
LIN {X 0,Y 608.53,Z 497.902,A -85,B 0,C 180,E1 -463.058,E2 -463.058} C_VEL
LIN {X 0,Y 608.518,Z 471.266,A -85,B 0,C 180,E1 -465.748,E2 -465.748} C_VEL
LIN {X 0,Y 608.538,Z 443.527,A -85,B 0,C 180,E1 -468.605,E2 -468.605} C_VEL
LIN {X 0,Y 608.638,Z 419.154,A -85,B 0,C 180,E1 -471.152,E2 -471.152} C_VEL
LIN {X 0,Y 608.7,Z 391.806,A -85,B 0,C 180,E1 -474.065,E2 -474.065} C_VEL
LIN {X 0,Y 608.68,Z 373.767,A -85,B 0,C 180,E1 -476.025,E2 -476.025} C_VEL
LIN {X 0,Y 608.468,Z 372.744,A -85,B 0,C 180,E1 -476.196,E2 -476.196} C_VEL
LIN {X 0,Y 608.385,Z 372.696,A -85,B 0,C 180,E1 -479.024,E2 -479.024} C_VEL
LIN {X 0,Y 608.391,Z 372.697,A -85,B 0,C 180,E1 -481.321,E2 -481.321} C_VEL
LIN {X 0,Y 608.426,Z 372.698,A -85,B 0,C 180,E1 -483.728,E2 -483.728} C_VEL
LIN {X 0,Y 608.44,Z 372.696,A -85,B 0,C 180,E1 -486.093,E2 -486.093} C_VEL
LIN {X 0,Y 608.398,Z 372.695,A -85,B 0,C 180,E1 -488.594,E2 -488.594} C_VEL
LIN {X 0,Y 608.402,Z 372.695,A -85,B 0,C 180,E1 -491.181,E2 -491.181} C_VEL
LIN {X 0,Y 608.466,Z 372.695,A -85,B 0,C 180,E1 -493.87,E2 -493.87} C_VEL
LIN {X 0,Y 608.428,Z 372.69,A -85,B 0,C 180,E1 -496.696,E2 -496.696} C_VEL
LIN {X 0,Y 608.406,Z 372.693,A -85,B 0,C 180,E1 -498.819,E2 -498.819} C_VEL
LIN {X 0,Y 608.417,Z 372.698,A -85,B 0,C 180,E1 -501.408,E2 -501.408} C_VEL
LIN {X 0,Y 608.447,Z 372.693,A -85,B 0,C 180,E1 -503.955,E2 -503.955} C_VEL
LIN {X 0,Y 608.445,Z 372.689,A -85,B 0,C 180,E1 -506.328,E2 -506.328} C_VEL
LIN {X 0,Y 608.435,Z 372.69,A -85,B 0,C 180,E1 -508.735,E2 -508.735} C_VEL
LIN {X 0,Y 608.472,Z 372.694,A -85,B 0,C 180,E1 -511.381,E2 -511.381} C_VEL
LIN {X 0,Y 608.456,Z 372.687,A -85,B 0,C 180,E1 -514.283,E2 -514.283} C_VEL
LIN {X 0,Y 608.435,Z 372.692,A -85,B 0,C 180,E1 -516.875,E2 -516.875} C_VEL
LIN {X 0,Y 608.464,Z 372.69,A -85,B 0,C 180,E1 -519.726,E2 -519.726} C_VEL
LIN {X 0,Y 608.454,Z 372.69,A -85,B 0,C 180,E1 -521.828,E2 -521.828} C_VEL
LIN {X 0,Y 608.456,Z 372.688,A -85,B 0,C 180,E1 -524.594,E2 -524.594} C_VEL
LIN {X 0,Y 608.488,Z 372.839,A -85,B 0,C 180,E1 -527.196,E2 -527.196} C_VEL
LIN {X 0,Y 608.595,Z 373.911,A -85,B 0,C 180,E1 -527.304,E2 -527.304} C_VEL
LIN {X 0,Y 608.558,Z 457.764,A -85,B 0,C 180,E1 -528.319,E2 -528.319} C_VEL
LIN {X 0,Y 608.539,Z 471.123,A -85,B 0,C 180,E1 -528.614,E2 -528.614} C_VEL
LIN {X 0,Y 608.529,Z 484.356,A -85,B 0,C 180,E1 -529.055,E2 -529.055} C_VEL
LIN {X 0,Y 608.508,Z 496.36,A -85,B 0,C 180,E1 -529.603,E2 -529.603} C_VEL
LIN {X 0,Y 608.504,Z 507.785,A -85,B 0,C 180,E1 -530.275,E2 -530.275} C_VEL
LIN {X 0,Y 608.474,Z 518.082,A -85,B 0,C 180,E1 -531.029,E2 -531.029} C_VEL
LIN {X 0,Y 608.464,Z 527.35,A -85,B 0,C 180,E1 -531.866,E2 -531.866} C_VEL
LIN {X 0,Y 608.466,Z 536.323,A -85,B 0,C 180,E1 -532.867,E2 -532.867} C_VEL
LIN {X 0,Y 608.444,Z 543.552,A -85,B 0,C 180,E1 -533.867,E2 -533.867} C_VEL
LIN {X 0,Y 608.462,Z 548.432,A -85,B 0,C 180,E1 -534.698,E2 -534.698} C_VEL
LIN {X 0,Y 608.439,Z 553.176,A -85,B 0,C 180,E1 -535.694,E2 -535.694} C_VEL
LIN {X 0,Y 608.425,Z 556.811,A -85,B 0,C 180,E1 -536.689,E2 -536.689} C_VEL
LIN {X 0,Y 608.425,Z 558.691,A -85,B 0,C 180,E1 -537.352,E2 -537.352} C_VEL
LIN {X 0,Y 608.444,Z 560.127,A -85,B 0,C 180,E1 -538.014,E2 -538.014} C_VEL
LIN {X 0,Y 608.439,Z 561.752,A -85,B 0,C 180,E1 -539.338,E2 -539.338} C_VEL
LIN {X 0,Y 608.435,Z 561.995,A -85,B 0,C 180,E1 -540,E2 -540} C_VEL
LIN {X 0,Y 608.438,Z 561.815,A -85,B 0,C 180,E1 -540.662,E2 -540.662} C_VEL
LIN {X 0,Y 608.444,Z 560.276,A -85,B 0,C 180,E1 -541.986,E2 -541.986} C_VEL
LIN {X 0,Y 608.426,Z 558.916,A -85,B 0,C 180,E1 -542.648,E2 -542.648} C_VEL
LIN {X 0,Y 608.449,Z 556.04,A -85,B 0,C 180,E1 -543.642,E2 -543.642} C_VEL
LIN {X 0,Y 608.433,Z 552.14,A -85,B 0,C 180,E1 -544.638,E2 -544.638} C_VEL
LIN {X 0,Y 608.449,Z 547.109,A -85,B 0,C 180,E1 -545.634,E2 -545.634} C_VEL
LIN {X 0,Y 608.441,Z 540.794,A -85,B 0,C 180,E1 -546.633,E2 -546.633} C_VEL
LIN {X 0,Y 608.475,Z 532.878,A -85,B 0,C 180,E1 -547.633,E2 -547.633} C_VEL
LIN {X 0,Y 608.472,Z 523.029,A -85,B 0,C 180,E1 -548.636,E2 -548.636} C_VEL
LIN {X 0,Y 608.477,Z 520.936,A -85,B 0,C 180,E1 -548.819,E2 -548.819} C_VEL
LIN {X 0,Y 607.81,Z 516.599,A -85,B 0,C 180,E1 -549.19,E2 -549.19} C_VEL
LIN {X 0,Y 604.969,Z 509.341,A -85,B 0,C 180,E1 -549.77,E2 -549.77} C_VEL
LIN {X 0,Y 602.151,Z 501.705,A -85,B 0,C 180,E1 -550.301,E2 -550.301} C_VEL
LIN {X 0,Y 601.522,Z 496.637,A -85,B 0,C 180,E1 -550.594,E2 -550.594} C_VEL
LIN {X 0,Y 601.548,Z 484.755,A -85,B 0,C 180,E1 -551.148,E2 -551.148} C_VEL
LIN {X 0,Y 601.607,Z 471.315,A -85,B 0,C 180,E1 -551.604,E2 -551.604} C_VEL
LIN {X 0,Y 601.614,Z 458.025,A -85,B 0,C 180,E1 -551.903,E2 -551.903} C_VEL
LIN {X 0,Y 601.639,Z 374.643,A -85,B 0,C 180,E1 -552.931,E2 -552.931} C_VEL
LIN {X 0,Y 601.428,Z 373.636,A -85,B 0,C 180,E1 -553.064,E2 -553.064} C_VEL
LIN {X 0,Y 601.408,Z 373.566,A -85,B 0,C 180,E1 -555.592,E2 -555.592} C_VEL
LIN {X 0,Y 601.423,Z 373.567,A -85,B 0,C 180,E1 -558.392,E2 -558.392} C_VEL
LIN {X 0,Y 601.405,Z 373.569,A -85,B 0,C 180,E1 -561.239,E2 -561.239} C_VEL
LIN {X 0,Y 601.462,Z 373.56,A -85,B 0,C 180,E1 -564.14,E2 -564.14} C_VEL
LIN {X 0,Y 601.426,Z 373.567,A -85,B 0,C 180,E1 -567.113,E2 -567.113} C_VEL
LIN {X 0,Y 601.415,Z 373.565,A -85,B 0,C 180,E1 -569.393,E2 -569.393} C_VEL
LIN {X 0,Y 601.401,Z 373.566,A -85,B 0,C 180,E1 -571.727,E2 -571.727} C_VEL
LIN {X 0,Y 601.424,Z 373.564,A -85,B 0,C 180,E1 -574.119,E2 -574.119} C_VEL
LIN {X 0,Y 601.398,Z 373.575,A -85,B 0,C 180,E1 -576.584,E2 -576.584} C_VEL
LIN {X 0,Y 601.402,Z 373.569,A -85,B 0,C 180,E1 -579.128,E2 -579.128} C_VEL
LIN {X 0,Y 601.422,Z 373.563,A -85,B 0,C 180,E1 -581.766,E2 -581.766} C_VEL
LIN {X 0,Y 601.4,Z 373.575,A -85,B 0,C 180,E1 -584.533,E2 -584.533} C_VEL
LIN {X 0,Y 601.432,Z 373.569,A -85,B 0,C 180,E1 -586.427,E2 -586.427} C_VEL
LIN {X 0,Y 601.407,Z 373.568,A -85,B 0,C 180,E1 -589.125,E2 -589.125} C_VEL
LIN {X 0,Y 601.411,Z 373.564,A -85,B 0,C 180,E1 -591.731,E2 -591.731} C_VEL
LIN {X 0,Y 601.388,Z 373.573,A -85,B 0,C 180,E1 -594.245,E2 -594.245} C_VEL
LIN {X 0,Y 601.425,Z 373.571,A -85,B 0,C 180,E1 -596.686,E2 -596.686} C_VEL
LIN {X 0,Y 601.398,Z 373.569,A -85,B 0,C 180,E1 -599.057,E2 -599.057} C_VEL
LIN {X 0,Y 601.405,Z 373.566,A -85,B 0,C 180,E1 -601.372,E2 -601.372} C_VEL
LIN {X 0,Y 601.464,Z 373.79,A -85,B 0,C 180,E1 -604.202,E2 -604.202} C_VEL
LIN {X 0,Y 601.915,Z 376.884,A -85,B 0,C 180,E1 -604.59,E2 -604.59} C_VEL
LIN {X 0,Y 601.813,Z 403.144,A -85,B 0,C 180,E1 -607.57,E2 -607.57} C_VEL
LIN {X 0,Y 601.693,Z 428.411,A -85,B 0,C 180,E1 -610.378,E2 -610.378} C_VEL
LIN {X 0,Y 601.539,Z 453.618,A -85,B 0,C 180,E1 -613.131,E2 -613.131} C_VEL
LIN {X 0,Y 601.519,Z 480.281,A -85,B 0,C 180,E1 -616.006,E2 -616.006} C_VEL
LIN {X 0,Y 601.514,Z 488.134,A -85,B 0,C 180,E1 -616.83,E2 -616.83} C_VEL
LIN {X 0,Y 601.688,Z 493.549,A -85,B 0,C 180,E1 -616.92,E2 -616.92} C_VEL
LIN {X 0,Y 601.626,Z 597.817,A -85,B 0,C 180,E1 -618.183,E2 -618.183} C_VEL
LIN {X 0,Y 601.576,Z 611.111,A -85,B 0,C 180,E1 -618.481,E2 -618.481} C_VEL
LIN {X 0,Y 601.544,Z 623.479,A -85,B 0,C 180,E1 -618.892,E2 -618.892} C_VEL
LIN {X 0,Y 601.522,Z 634.748,A -85,B 0,C 180,E1 -619.396,E2 -619.396} C_VEL
LIN {X 0,Y 601.484,Z 646.511,A -85,B 0,C 180,E1 -620.076,E2 -620.076} C_VEL
LIN {X 0,Y 601.444,Z 657.018,A -85,B 0,C 180,E1 -620.839,E2 -620.839} C_VEL
LIN {X 0,Y 601.429,Z 665.63,A -85,B 0,C 180,E1 -621.601,E2 -621.601} C_VEL
LIN {X 0,Y 601.418,Z 673.563,A -85,B 0,C 180,E1 -622.446,E2 -622.446} C_VEL
LIN {X 0,Y 601.377,Z 680.89,A -85,B 0,C 180,E1 -623.393,E2 -623.393} C_VEL
LIN {X 0,Y 601.372,Z 686.613,A -85,B 0,C 180,E1 -624.299,E2 -624.299} C_VEL
LIN {X 0,Y 601.335,Z 691.753,A -85,B 0,C 180,E1 -625.307,E2 -625.307} C_VEL
LIN {X 0,Y 601.367,Z 695.742,A -85,B 0,C 180,E1 -626.315,E2 -626.315} C_VEL
LIN {X 0,Y 601.324,Z 698.695,A -85,B 0,C 180,E1 -627.321,E2 -627.321} C_VEL
LIN {X 0,Y 601.342,Z 700.13,A -85,B 0,C 180,E1 -627.991,E2 -627.991} C_VEL
LIN {X 0,Y 601.339,Z 701.753,A -85,B 0,C 180,E1 -629.33,E2 -629.33} C_VEL
LIN {X 0,Y 601.336,Z 701.996,A -85,B 0,C 180,E1 -630,E2 -630} C_VEL
LIN {X 0,Y 601.339,Z 701.816,A -85,B 0,C 180,E1 -630.67,E2 -630.67} C_VEL
LIN {X 0,Y 601.343,Z 700.277,A -85,B 0,C 180,E1 -632.009,E2 -632.009} C_VEL
LIN {X 0,Y 601.326,Z 698.91,A -85,B 0,C 180,E1 -632.68,E2 -632.68} C_VEL
LIN {X 0,Y 601.368,Z 696.033,A -85,B 0,C 180,E1 -633.685,E2 -633.685} C_VEL
LIN {X 0,Y 601.337,Z 692.136,A -85,B 0,C 180,E1 -634.693,E2 -634.693} C_VEL
LIN {X 0,Y 601.373,Z 687.108,A -85,B 0,C 180,E1 -635.701,E2 -635.701} C_VEL
LIN {X 0,Y 601.382,Z 680.79,A -85,B 0,C 180,E1 -636.711,E2 -636.711} C_VEL
LIN {X 0,Y 601.396,Z 672.867,A -85,B 0,C 180,E1 -637.724,E2 -637.724} C_VEL
LIN {X 0,Y 601.421,Z 664.796,A -85,B 0,C 180,E1 -638.569,E2 -638.569} C_VEL
LIN {X 0,Y 601.453,Z 654.962,A -85,B 0,C 180,E1 -639.416,E2 -639.416} C_VEL
LIN {X 0,Y 601.5,Z 643.916,A -85,B 0,C 180,E1 -640.179,E2 -640.179} C_VEL
LIN {X 0,Y 601.522,Z 631.907,A -85,B 0,C 180,E1 -640.832,E2 -640.832} C_VEL
LIN {X 0,Y 601.57,Z 620.394,A -85,B 0,C 180,E1 -641.314,E2 -641.314} C_VEL
LIN {X 0,Y 601.604,Z 607.291,A -85,B 0,C 180,E1 -641.711,E2 -641.711} C_VEL
LIN {X 0,Y 601.628,Z 593.764,A -85,B 0,C 180,E1 -641.967,E2 -641.967} C_VEL
LIN {X 0,Y 601.569,Z 488.768,A -85,B 0,C 180,E1 -643.233,E2 -643.233} C_VEL
LIN {X 0,Y 601.486,Z 487.226,A -85,B 0,C 180,E1 -643.342,E2 -643.342} C_VEL
LIN {X 0,Y 601.566,Z 461.448,A -85,B 0,C 180,E1 -646.109,E2 -646.109} C_VEL
LIN {X 0,Y 601.642,Z 435.064,A -85,B 0,C 180,E1 -648.981,E2 -648.981} C_VEL
LIN {X 0,Y 601.746,Z 409.891,A -85,B 0,C 180,E1 -651.766,E2 -651.766} C_VEL
LIN {X 0,Y 601.884,Z 383.951,A -85,B 0,C 180,E1 -654.692,E2 -654.692} C_VEL
LIN {X 0,Y 601.888,Z 376.054,A -85,B 0,C 180,E1 -655.597,E2 -655.597} C_VEL
LIN {X 0,Y 601.419,Z 373.63,A -85,B 0,C 180,E1 -655.94,E2 -655.94} C_VEL
LIN {X 0,Y 601.403,Z 373.566,A -85,B 0,C 180,E1 -658.782,E2 -658.782} C_VEL
LIN {X 0,Y 601.416,Z 373.572,A -85,B 0,C 180,E1 -661.453,E2 -661.453} C_VEL
LIN {X 0,Y 601.42,Z 373.566,A -85,B 0,C 180,E1 -664.119,E2 -664.119} C_VEL
LIN {X 0,Y 601.378,Z 373.568,A -85,B 0,C 180,E1 -666.585,E2 -666.585} C_VEL
LIN {X 0,Y 601.387,Z 373.57,A -85,B 0,C 180,E1 -669.129,E2 -669.129} C_VEL
LIN {X 0,Y 601.418,Z 373.572,A -85,B 0,C 180,E1 -671.766,E2 -671.766} C_VEL
LIN {X 0,Y 601.402,Z 373.565,A -85,B 0,C 180,E1 -674.533,E2 -674.533} C_VEL
LIN {X 0,Y 601.391,Z 373.573,A -85,B 0,C 180,E1 -677.412,E2 -677.412} C_VEL
LIN {X 0,Y 601.398,Z 373.571,A -85,B 0,C 180,E1 -680.004,E2 -680.004} C_VEL
LIN {X 0,Y 601.393,Z 373.566,A -85,B 0,C 180,E1 -682.624,E2 -682.624} C_VEL
LIN {X 0,Y 601.376,Z 373.57,A -85,B 0,C 180,E1 -685.065,E2 -685.065} C_VEL
LIN {X 0,Y 601.421,Z 373.57,A -85,B 0,C 180,E1 -687.483,E2 -687.483} C_VEL
LIN {X 0,Y 601.411,Z 373.572,A -85,B 0,C 180,E1 -689.855,E2 -689.855} C_VEL
LIN {X 0,Y 601.374,Z 373.569,A -85,B 0,C 180,E1 -692.646,E2 -692.646} C_VEL
LIN {X 0,Y 601.377,Z 373.57,A -85,B 0,C 180,E1 -695.12,E2 -695.12} C_VEL
LIN {X 0,Y 601.419,Z 373.568,A -85,B 0,C 180,E1 -697.395,E2 -697.395} C_VEL
LIN {X 0,Y 601.387,Z 373.57,A -85,B 0,C 180,E1 -700.19,E2 -700.19} C_VEL
LIN {X 0,Y 601.375,Z 373.569,A -85,B 0,C 180,E1 -703.012,E2 -703.012} C_VEL
LIN {X 0,Y 601.422,Z 373.57,A -85,B 0,C 180,E1 -705.91,E2 -705.91} C_VEL
LIN {X 0,Y 601.399,Z 373.565,A -85,B 0,C 180,E1 -708.541,E2 -708.541} C_VEL
LIN {X 0,Y 601.39,Z 373.57,A -85,B 0,C 180,E1 -711.262,E2 -711.262} C_VEL
LIN {X 0,Y 601.406,Z 373.571,A -85,B 0,C 180,E1 -713.963,E2 -713.963} C_VEL
LIN {X 0,Y 601.358,Z 373.57,A -85,B 0,C 180,E1 -716.65,E2 -716.65} C_VEL
LIN {X 0,Y 601.379,Z 373.568,A -85,B 0,C 180,E1 -718.661,E2 -718.661} C_VEL
LIN {X 0,Y 601.366,Z 373.57,A -85,B 0,C 180,E1 -720.67,E2 -720.67} C_VEL
LIN {X 0,Y 601.398,Z 373.565,A -85,B 0,C 180,E1 -722.679,E2 -722.679} C_VEL
LIN {X 0,Y 601.395,Z 373.57,A -85,B 0,C 180,E1 -725.364,E2 -725.364} C_VEL
LIN {X 0,Y 601.435,Z 373.567,A -85,B 0,C 180,E1 -728.061,E2 -728.061} C_VEL
LIN {X 0,Y 601.379,Z 373.568,A -85,B 0,C 180,E1 -730.987,E2 -730.987} C_VEL
LIN {X 0,Y 601.395,Z 373.572,A -85,B 0,C 180,E1 -733.516,E2 -733.516} C_VEL
LIN {X 0,Y 601.405,Z 373.567,A -85,B 0,C 180,E1 -736.288,E2 -736.288} C_VEL
LIN {X 0,Y 601.366,Z 373.571,A -85,B 0,C 180,E1 -739.101,E2 -739.101} C_VEL
LIN {X 0,Y 601.381,Z 373.57,A -85,B 0,C 180,E1 -741.24,E2 -741.24} C_VEL
LIN {X 0,Y 601.429,Z 373.567,A -85,B 0,C 180,E1 -744.142,E2 -744.142} C_VEL
LIN {X 0,Y 601.372,Z 373.571,A -85,B 0,C 180,E1 -746.365,E2 -746.365} C_VEL
LIN {X 0,Y 601.391,Z 373.57,A -85,B 0,C 180,E1 -749.395,E2 -749.395} C_VEL
LIN {X 0,Y 601.388,Z 373.576,A -85,B 0,C 180,E1 -751.728,E2 -751.728} C_VEL
LIN {X 0,Y 601.407,Z 373.57,A -85,B 0,C 180,E1 -754.12,E2 -754.12} C_VEL
LIN {X 0,Y 601.368,Z 373.57,A -85,B 0,C 180,E1 -756.586,E2 -756.586} C_VEL
LIN {X 0,Y 601.394,Z 373.571,A -85,B 0,C 180,E1 -759.53,E2 -759.53} C_VEL
LIN {X 0,Y 601.41,Z 373.572,A -85,B 0,C 180,E1 -761.766,E2 -761.766} C_VEL
LIN {X 0,Y 601.369,Z 373.571,A -85,B 0,C 180,E1 -764.529,E2 -764.529} C_VEL
LIN {X 0,Y 601.404,Z 373.567,A -85,B 0,C 180,E1 -766.43,E2 -766.43} C_VEL
LIN {X 0,Y 601.351,Z 373.571,A -85,B 0,C 180,E1 -769.12,E2 -769.12} C_VEL
LIN {X 0,Y 601.383,Z 373.576,A -85,B 0,C 180,E1 -771.729,E2 -771.729} C_VEL
LIN {X 0,Y 601.371,Z 373.574,A -85,B 0,C 180,E1 -774.244,E2 -774.244} C_VEL
LIN {X 0,Y 601.38,Z 373.569,A -85,B 0,C 180,E1 -776.683,E2 -776.683} C_VEL
LIN {X 0,Y 601.364,Z 373.571,A -85,B 0,C 180,E1 -779.055,E2 -779.055} C_VEL
LIN {X 0,Y 601.365,Z 373.573,A -85,B 0,C 180,E1 -781.369,E2 -781.369} C_VEL
LIN {X 0,Y 601.402,Z 373.74,A -85,B 0,C 180,E1 -783.613,E2 -783.613} C_VEL
LIN {X 0,Y 601.979,Z 377.006,A -85,B 0,C 180,E1 -784.022,E2 -784.022} C_VEL
LIN {X 0,Y 601.823,Z 400.661,A -85,B 0,C 180,E1 -786.606,E2 -786.606} C_VEL
LIN {X 0,Y 601.74,Z 424.136,A -85,B 0,C 180,E1 -789.125,E2 -789.125} C_VEL
LIN {X 0,Y 601.634,Z 451.092,A -85,B 0,C 180,E1 -791.967,E2 -791.967} C_VEL
LIN {X 0,Y 601.517,Z 474.626,A -85,B 0,C 180,E1 -794.411,E2 -794.411} C_VEL
LIN {X 0,Y 601.521,Z 497.897,A -85,B 0,C 180,E1 -796.787,E2 -796.787} C_VEL
LIN {X 0,Y 601.67,Z 503.704,A -85,B 0,C 180,E1 -796.877,E2 -796.877} C_VEL
LIN {X 0,Y 601.614,Z 607.937,A -85,B 0,C 180,E1 -798.139,E2 -798.139} C_VEL
LIN {X 0,Y 601.589,Z 621.211,A -85,B 0,C 180,E1 -798.438,E2 -798.438} C_VEL
LIN {X 0,Y 601.549,Z 632.919,A -85,B 0,C 180,E1 -798.826,E2 -798.826} C_VEL
LIN {X 0,Y 601.53,Z 643.92,A -85,B 0,C 180,E1 -799.311,E2 -799.311} C_VEL
LIN {X 0,Y 601.486,Z 654.577,A -85,B 0,C 180,E1 -799.906,E2 -799.906} C_VEL
LIN {X 0,Y 601.448,Z 665.474,A -85,B 0,C 180,E1 -800.669,E2 -800.669} C_VEL
LIN {X 0,Y 601.429,Z 676.11,A -85,B 0,C 180,E1 -801.601,E2 -801.601} C_VEL
LIN {X 0,Y 601.418,Z 683.959,A -85,B 0,C 180,E1 -802.446,E2 -802.446} C_VEL
LIN {X 0,Y 601.37,Z 691.224,A -85,B 0,C 180,E1 -803.398,E2 -803.398} C_VEL
LIN {X 0,Y 601.372,Z 696.865,A -85,B 0,C 180,E1 -804.299,E2 -804.299} C_VEL
LIN {X 0,Y 601.336,Z 701.949,A -85,B 0,C 180,E1 -805.307,E2 -805.307} C_VEL
LIN {X 0,Y 601.368,Z 705.896,A -85,B 0,C 180,E1 -806.315,E2 -806.315} C_VEL
LIN {X 0,Y 601.325,Z 708.809,A -85,B 0,C 180,E1 -807.32,E2 -807.32} C_VEL
LIN {X 0,Y 601.343,Z 710.201,A -85,B 0,C 180,E1 -807.991,E2 -807.991} C_VEL
LIN {X 0,Y 601.339,Z 711.784,A -85,B 0,C 180,E1 -809.33,E2 -809.33} C_VEL
LIN {X 0,Y 601.335,Z 712,A -85,B 0,C 180,E1 -810,E2 -810} C_VEL
LIN {X 0,Y 601.347,Z 711.184,A -85,B 0,C 180,E1 -811.339,E2 -811.339} C_VEL
LIN {X 0,Y 601.343,Z 710.202,A -85,B 0,C 180,E1 -812.009,E2 -812.009} C_VEL
LIN {X 0,Y 601.325,Z 708.81,A -85,B 0,C 180,E1 -812.679,E2 -812.679} C_VEL
LIN {X 0,Y 601.368,Z 705.896,A -85,B 0,C 180,E1 -813.685,E2 -813.685} C_VEL
LIN {X 0,Y 601.336,Z 701.95,A -85,B 0,C 180,E1 -814.693,E2 -814.693} C_VEL
LIN {X 0,Y 601.372,Z 695.877,A -85,B 0,C 180,E1 -815.869,E2 -815.869} C_VEL
LIN {X 0,Y 601.382,Z 689.236,A -85,B 0,C 180,E1 -816.88,E2 -816.88} C_VEL
LIN {X 0,Y 601.401,Z 680.99,A -85,B 0,C 180,E1 -817.892,E2 -817.892} C_VEL
LIN {X 0,Y 601.436,Z 672.537,A -85,B 0,C 180,E1 -818.738,E2 -818.738} C_VEL
LIN {X 0,Y 601.448,Z 662.092,A -85,B 0,C 180,E1 -819.585,E2 -819.585} C_VEL
LIN {X 0,Y 601.481,Z 651.758,A -85,B 0,C 180,E1 -820.264,E2 -820.264} C_VEL
LIN {X 0,Y 601.538,Z 640.896,A -85,B 0,C 180,E1 -820.836,E2 -820.836} C_VEL
LIN {X 0,Y 601.566,Z 628.373,A -85,B 0,C 180,E1 -821.34,E2 -821.34} C_VEL
LIN {X 0,Y 601.603,Z 615.352,A -85,B 0,C 180,E1 -821.711,E2 -821.711} C_VEL
LIN {X 0,Y 601.619,Z 602.085,A -85,B 0,C 180,E1 -821.946,E2 -821.946} C_VEL
LIN {X 0,Y 601.579,Z 498.535,A -85,B 0,C 180,E1 -823.19,E2 -823.19} C_VEL
LIN {X 0,Y 601.521,Z 497.345,A -85,B 0,C 180,E1 -823.255,E2 -823.255} C_VEL
LIN {X 0,Y 601.571,Z 469.585,A -85,B 0,C 180,E1 -826.109,E2 -826.109} C_VEL
LIN {X 0,Y 601.644,Z 443.003,A -85,B 0,C 180,E1 -828.881,E2 -828.881} C_VEL
LIN {X 0,Y 601.766,Z 417.473,A -85,B 0,C 180,E1 -831.585,E2 -831.585} C_VEL
LIN {X 0,Y 601.899,Z 392.715,A -85,B 0,C 180,E1 -834.255,E2 -834.255} C_VEL
LIN {X 0,Y 601.958,Z 376.006,A -85,B 0,C 180,E1 -836.089,E2 -836.089} C_VEL
LIN {X 0,Y 601.411,Z 373.661,A -85,B 0,C 180,E1 -836.41,E2 -836.41} C_VEL
LIN {X 0,Y 601.374,Z 373.572,A -85,B 0,C 180,E1 -839.396,E2 -839.396} C_VEL
LIN {X 0,Y 601.369,Z 373.577,A -85,B 0,C 180,E1 -841.729,E2 -841.729} C_VEL
LIN {X 0,Y 601.397,Z 373.574,A -85,B 0,C 180,E1 -844.121,E2 -844.121} C_VEL
LIN {X 0,Y 601.366,Z 373.572,A -85,B 0,C 180,E1 -846.586,E2 -846.586} C_VEL
LIN {X 0,Y 601.397,Z 373.572,A -85,B 0,C 180,E1 -849.53,E2 -849.53} C_VEL
LIN {X 0,Y 601.413,Z 373.574,A -85,B 0,C 180,E1 -851.766,E2 -851.766} C_VEL
LIN {X 0,Y 601.4,Z 373.567,A -85,B 0,C 180,E1 -854.533,E2 -854.533} C_VEL
LIN {X 0,Y 601.385,Z 373.573,A -85,B 0,C 180,E1 -857.412,E2 -857.412} C_VEL
LIN {X 0,Y 601.397,Z 373.571,A -85,B 0,C 180,E1 -860.004,E2 -860.004} C_VEL
LIN {X 0,Y 601.397,Z 373.566,A -85,B 0,C 180,E1 -862.623,E2 -862.623} C_VEL
LIN {X 0,Y 601.385,Z 373.57,A -85,B 0,C 180,E1 -865.066,E2 -865.066} C_VEL
LIN {X 0,Y 601.434,Z 373.571,A -85,B 0,C 180,E1 -867.484,E2 -867.484} C_VEL
LIN {X 0,Y 601.431,Z 373.567,A -85,B 0,C 180,E1 -869.852,E2 -869.852} C_VEL
LIN {X 0,Y 601.386,Z 373.568,A -85,B 0,C 180,E1 -872.644,E2 -872.644} C_VEL
LIN {X 0,Y 601.39,Z 373.573,A -85,B 0,C 180,E1 -875.121,E2 -875.121} C_VEL
LIN {X 0,Y 601.419,Z 373.574,A -85,B 0,C 180,E1 -877.395,E2 -877.395} C_VEL
LIN {X 0,Y 601.399,Z 373.567,A -85,B 0,C 180,E1 -880.19,E2 -880.19} C_VEL
LIN {X 0,Y 601.43,Z 373.569,A -85,B 0,C 180,E1 -883.014,E2 -883.014} C_VEL
LIN {X 0,Y 601.426,Z 373.566,A -85,B 0,C 180,E1 -885.908,E2 -885.908} C_VEL
LIN {X 0,Y 601.443,Z 373.764,A -85,B 0,C 180,E1 -887.065,E2 -887.065} C_VEL
LIN {X 0,Y 601.669,Z 374.797,A -85,B 0,C 180,E1 -887.166,E2 -887.166} C_VEL
LIN {X 0,Y 601.63,Z 457.729,A -85,B 0,C 180,E1 -888.183,E2 -888.183} C_VEL
LIN {X 0,Y 601.599,Z 470.394,A -85,B 0,C 180,E1 -888.46,E2 -888.46} C_VEL
LIN {X 0,Y 601.566,Z 484.229,A -85,B 0,C 180,E1 -888.921,E2 -888.921} C_VEL
LIN {X 0,Y 601.514,Z 496.351,A -85,B 0,C 180,E1 -889.481,E2 -889.481} C_VEL
LIN {X 0,Y 601.472,Z 507.789,A -85,B 0,C 180,E1 -890.161,E2 -890.161} C_VEL
LIN {X 0,Y 601.438,Z 518.088,A -85,B 0,C 180,E1 -890.924,E2 -890.924} C_VEL
LIN {X 0,Y 601.411,Z 527.355,A -85,B 0,C 180,E1 -891.77,E2 -891.77} C_VEL
LIN {X 0,Y 601.388,Z 536.326,A -85,B 0,C 180,E1 -892.783,E2 -892.783} C_VEL
LIN {X 0,Y 601.376,Z 543.454,A -85,B 0,C 180,E1 -893.781,E2 -893.781} C_VEL
LIN {X 0,Y 601.372,Z 548.43,A -85,B 0,C 180,E1 -894.635,E2 -894.635} C_VEL
LIN {X 0,Y 601.354,Z 553.17,A -85,B 0,C 180,E1 -895.643,E2 -895.643} C_VEL
LIN {X 0,Y 601.344,Z 556.808,A -85,B 0,C 180,E1 -896.65,E2 -896.65} C_VEL
LIN {X 0,Y 601.324,Z 558.693,A -85,B 0,C 180,E1 -897.32,E2 -897.32} C_VEL
LIN {X 0,Y 601.343,Z 560.129,A -85,B 0,C 180,E1 -897.991,E2 -897.991} C_VEL
LIN {X 0,Y 601.339,Z 561.753,A -85,B 0,C 180,E1 -899.33,E2 -899.33} C_VEL
LIN {X 0,Y 601.336,Z 561.996,A -85,B 0,C 180,E1 -900,E2 -900} C_VEL
LIN {X 0,Y 601.339,Z 561.815,A -85,B 0,C 180,E1 -900.67,E2 -900.67} C_VEL
LIN {X 0,Y 601.343,Z 560.277,A -85,B 0,C 180,E1 -902.009,E2 -902.009} C_VEL
LIN {X 0,Y 601.325,Z 558.904,A -85,B 0,C 180,E1 -902.68,E2 -902.68} C_VEL
LIN {X 0,Y 601.368,Z 556.029,A -85,B 0,C 180,E1 -903.685,E2 -903.685} C_VEL
LIN {X 0,Y 601.336,Z 552.129,A -85,B 0,C 180,E1 -904.693,E2 -904.693} C_VEL
LIN {X 0,Y 601.373,Z 547.101,A -85,B 0,C 180,E1 -905.701,E2 -905.701} C_VEL
LIN {X 0,Y 601.382,Z 540.789,A -85,B 0,C 180,E1 -906.711,E2 -906.711} C_VEL
LIN {X 0,Y 601.396,Z 532.875,A -85,B 0,C 180,E1 -907.723,E2 -907.723} C_VEL
LIN {X 0,Y 601.422,Z 524.809,A -85,B 0,C 180,E1 -908.569,E2 -908.569} C_VEL
LIN {X 0,Y 601.452,Z 514.958,A -85,B 0,C 180,E1 -909.415,E2 -909.415} C_VEL
LIN {X 0,Y 601.496,Z 503.92,A -85,B 0,C 180,E1 -910.179,E2 -910.179} C_VEL
LIN {X 0,Y 601.522,Z 496.637,A -85,B 0,C 180,E1 -910.594,E2 -910.594} C_VEL
LIN {X 0,Y 600.897,Z 491.504,A -85,B 0,C 180,E1 -910.868,E2 -910.868} C_VEL
LIN {X 0,Y 598.098,Z 483.064,A -85,B 0,C 180,E1 -911.292,E2 -911.292} C_VEL
LIN {X 0,Y 595.289,Z 474.318,A -85,B 0,C 180,E1 -911.647,E2 -911.647} C_VEL
LIN {X 0,Y 594.641,Z 468.715,A -85,B 0,C 180,E1 -911.812,E2 -911.812} C_VEL
LIN {X 0,Y 594.693,Z 456.581,A -85,B 0,C 180,E1 -912.066,E2 -912.066} C_VEL
LIN {X 0,Y 594.659,Z 375.777,A -85,B 0,C 180,E1 -913.064,E2 -913.064} C_VEL
LIN {X 0,Y 594.412,Z 374.607,A -85,B 0,C 180,E1 -913.178,E2 -913.178} C_VEL
LIN {X 0,Y 594.363,Z 374.444,A -85,B 0,C 180,E1 -915.781,E2 -915.781} C_VEL
LIN {X 0,Y 594.386,Z 374.447,A -85,B 0,C 180,E1 -918.618,E2 -918.618} C_VEL
LIN {X 0,Y 594.366,Z 374.443,A -85,B 0,C 180,E1 -921.503,E2 -921.503} C_VEL
LIN {X 0,Y 594.393,Z 374.444,A -85,B 0,C 180,E1 -924.446,E2 -924.446} C_VEL
LIN {X 0,Y 594.373,Z 374.451,A -85,B 0,C 180,E1 -926.7,E2 -926.7} C_VEL
LIN {X 0,Y 594.384,Z 374.446,A -85,B 0,C 180,E1 -928.999,E2 -928.999} C_VEL
LIN {X 0,Y 594.377,Z 374.441,A -85,B 0,C 180,E1 -931.642,E2 -931.642} C_VEL
LIN {X 0,Y 594.38,Z 374.448,A -85,B 0,C 180,E1 -934.58,E2 -934.58} C_VEL
LIN {X 0,Y 594.389,Z 374.439,A -85,B 0,C 180,E1 -937.608,E2 -937.608} C_VEL
LIN {X 0,Y 594.37,Z 374.451,A -85,B 0,C 180,E1 -940.567,E2 -940.567} C_VEL
LIN {X 0,Y 594.353,Z 374.445,A -85,B 0,C 180,E1 -943.301,E2 -943.301} C_VEL
LIN {X 0,Y 594.363,Z 374.446,A -85,B 0,C 180,E1 -946.161,E2 -946.161} C_VEL
LIN {X 0,Y 594.371,Z 374.444,A -85,B 0,C 180,E1 -949.179,E2 -949.179} C_VEL
LIN {X 0,Y 594.381,Z 374.442,A -85,B 0,C 180,E1 -952.059,E2 -952.059} C_VEL
LIN {X 0,Y 594.348,Z 374.453,A -85,B 0,C 180,E1 -954.677,E2 -954.677} C_VEL
LIN {X 0,Y 594.376,Z 374.443,A -85,B 0,C 180,E1 -957.089,E2 -957.089} C_VEL
LIN {X 0,Y 594.372,Z 374.442,A -85,B 0,C 180,E1 -959.675,E2 -959.675} C_VEL
LIN {X 0,Y 594.378,Z 374.451,A -85,B 0,C 180,E1 -962.539,E2 -962.539} C_VEL
LIN {X 0,Y 594.394,Z 374.55,A -85,B 0,C 180,E1 -963.941,E2 -963.941} C_VEL
LIN {X 0,Y 595.119,Z 378.5,A -85,B 0,C 180,E1 -964.466,E2 -964.466} C_VEL
LIN {X 0,Y 594.956,Z 402.856,A -85,B 0,C 180,E1 -967.264,E2 -967.264} C_VEL
LIN {X 0,Y 594.804,Z 428.417,A -85,B 0,C 180,E1 -970.141,E2 -970.141} C_VEL
LIN {X 0,Y 594.59,Z 453.809,A -85,B 0,C 180,E1 -972.949,E2 -972.949} C_VEL
LIN {X 0,Y 594.54,Z 478.338,A -85,B 0,C 180,E1 -975.627,E2 -975.627} C_VEL
LIN {X 0,Y 594.54,Z 488.148,A -85,B 0,C 180,E1 -976.673,E2 -976.673} C_VEL
LIN {X 0,Y 594.787,Z 493.594,A -85,B 0,C 180,E1 -976.766,E2 -976.766} C_VEL
LIN {X 0,Y 594.68,Z 597.842,A -85,B 0,C 180,E1 -978.042,E2 -978.042} C_VEL
LIN {X 0,Y 594.645,Z 610.354,A -85,B 0,C 180,E1 -978.323,E2 -978.323} C_VEL
LIN {X 0,Y 594.57,Z 622.989,A -85,B 0,C 180,E1 -978.741,E2 -978.741} C_VEL
LIN {X 0,Y 594.537,Z 634.761,A -85,B 0,C 180,E1 -979.27,E2 -979.27} C_VEL
LIN {X 0,Y 594.484,Z 646.514,A -85,B 0,C 180,E1 -979.958,E2 -979.958} C_VEL
LIN {X 0,Y 594.414,Z 657.017,A -85,B 0,C 180,E1 -980.73,E2 -980.73} C_VEL
LIN {X 0,Y 594.366,Z 665.629,A -85,B 0,C 180,E1 -981.5,E2 -981.5} C_VEL
LIN {X 0,Y 594.347,Z 673.564,A -85,B 0,C 180,E1 -982.355,E2 -982.355} C_VEL
LIN {X 0,Y 594.305,Z 681.396,A -85,B 0,C 180,E1 -983.39,E2 -983.39} C_VEL
LIN {X 0,Y 594.289,Z 688.44,A -85,B 0,C 180,E1 -984.571,E2 -984.571} C_VEL
LIN {X 0,Y 594.27,Z 693.177,A -85,B 0,C 180,E1 -985.591,E2 -985.591} C_VEL
LIN {X 0,Y 594.267,Z 696.804,A -85,B 0,C 180,E1 -986.61,E2 -986.61} C_VEL
LIN {X 0,Y 594.225,Z 698.697,A -85,B 0,C 180,E1 -987.288,E2 -987.288} C_VEL
LIN {X 0,Y 594.241,Z 700.132,A -85,B 0,C 180,E1 -987.967,E2 -987.967} C_VEL
LIN {X 0,Y 594.24,Z 701.755,A -85,B 0,C 180,E1 -989.322,E2 -989.322} C_VEL
LIN {X 0,Y 594.236,Z 701.996,A -85,B 0,C 180,E1 -990,E2 -990} C_VEL
LIN {X 0,Y 594.239,Z 701.815,A -85,B 0,C 180,E1 -990.678,E2 -990.678} C_VEL
LIN {X 0,Y 594.242,Z 700.278,A -85,B 0,C 180,E1 -992.033,E2 -992.033} C_VEL
LIN {X 0,Y 594.226,Z 698.902,A -85,B 0,C 180,E1 -992.712,E2 -992.712} C_VEL
LIN {X 0,Y 594.289,Z 696.026,A -85,B 0,C 180,E1 -993.729,E2 -993.729} C_VEL
LIN {X 0,Y 594.241,Z 692.131,A -85,B 0,C 180,E1 -994.749,E2 -994.749} C_VEL
LIN {X 0,Y 594.299,Z 687.105,A -85,B 0,C 180,E1 -995.769,E2 -995.769} C_VEL
LIN {X 0,Y 594.316,Z 680.786,A -85,B 0,C 180,E1 -996.791,E2 -996.791} C_VEL
LIN {X 0,Y 594.347,Z 672.858,A -85,B 0,C 180,E1 -997.816,E2 -997.816} C_VEL
LIN {X 0,Y 594.366,Z 664.784,A -85,B 0,C 180,E1 -998.671,E2 -998.671} C_VEL
LIN {X 0,Y 594.415,Z 654.947,A -85,B 0,C 180,E1 -999.528,E2 -999.528} C_VEL
LIN {X 0,Y 594.473,Z 643.911,A -85,B 0,C 180,E1 -1000.301,E2 -1000.301} C_VEL
LIN {X 0,Y 594.551,Z 631.494,A -85,B 0,C 180,E1 -1000.981,E2 -1000.981} C_VEL
LIN {X 0,Y 594.612,Z 619.583,A -85,B 0,C 180,E1 -1001.477,E2 -1001.477} C_VEL
LIN {X 0,Y 594.638,Z 606.364,A -85,B 0,C 180,E1 -1001.872,E2 -1001.872} C_VEL
LIN {X 0,Y 594.679,Z 593.735,A -85,B 0,C 180,E1 -1002.109,E2 -1002.109} C_VEL
LIN {X 0,Y 594.674,Z 489.58,A -85,B 0,C 180,E1 -1003.376,E2 -1003.376} C_VEL
LIN {X 0,Y 594.493,Z 487.874,A -85,B 0,C 180,E1 -1003.437,E2 -1003.437} C_VEL
LIN {X 0,Y 594.599,Z 461.443,A -85,B 0,C 180,E1 -1006.303,E2 -1006.303} C_VEL
LIN {X 0,Y 594.754,Z 434.054,A -85,B 0,C 180,E1 -1009.322,E2 -1009.322} C_VEL
LIN {X 0,Y 594.904,Z 409.886,A -85,B 0,C 180,E1 -1012.03,E2 -1012.03} C_VEL
LIN {X 0,Y 595.107,Z 382.494,A -85,B 0,C 180,E1 -1015.16,E2 -1015.16} C_VEL
LIN {X 0,Y 595.054,Z 377.66,A -85,B 0,C 180,E1 -1015.725,E2 -1015.725} C_VEL
LIN {X 0,Y 594.37,Z 374.523,A -85,B 0,C 180,E1 -1016.161,E2 -1016.161} C_VEL
LIN {X 0,Y 594.373,Z 374.443,A -85,B 0,C 180,E1 -1018.999,E2 -1018.999} C_VEL
LIN {X 0,Y 594.373,Z 374.451,A -85,B 0,C 180,E1 -1021.641,E2 -1021.641} C_VEL
LIN {X 0,Y 594.361,Z 374.443,A -85,B 0,C 180,E1 -1024.582,E2 -1024.582} C_VEL
LIN {X 0,Y 594.365,Z 374.452,A -85,B 0,C 180,E1 -1027.605,E2 -1027.605} C_VEL
LIN {X 0,Y 594.355,Z 374.443,A -85,B 0,C 180,E1 -1030.569,E2 -1030.569} C_VEL
LIN {X 0,Y 594.342,Z 374.45,A -85,B 0,C 180,E1 -1033.302,E2 -1033.302} C_VEL
LIN {X 0,Y 594.346,Z 374.447,A -85,B 0,C 180,E1 -1036.163,E2 -1036.163} C_VEL
LIN {X 0,Y 594.364,Z 374.442,A -85,B 0,C 180,E1 -1038.534,E2 -1038.534} C_VEL
LIN {X 0,Y 594.366,Z 374.446,A -85,B 0,C 180,E1 -1041.298,E2 -1041.298} C_VEL
LIN {X 0,Y 594.347,Z 374.454,A -85,B 0,C 180,E1 -1043.755,E2 -1043.755} C_VEL
LIN {X 0,Y 594.363,Z 374.444,A -85,B 0,C 180,E1 -1046.238,E2 -1046.238} C_VEL
LIN {X 0,Y 594.36,Z 374.443,A -85,B 0,C 180,E1 -1048.649,E2 -1048.649} C_VEL
LIN {X 0,Y 594.343,Z 374.446,A -85,B 0,C 180,E1 -1051.05,E2 -1051.05} C_VEL
LIN {X 0,Y 594.36,Z 374.447,A -85,B 0,C 180,E1 -1054.055,E2 -1054.055} C_VEL
LIN {X 0,Y 594.368,Z 374.443,A -85,B 0,C 180,E1 -1056.295,E2 -1056.295} C_VEL
LIN {X 0,Y 594.389,Z 374.442,A -85,B 0,C 180,E1 -1059.224,E2 -1059.224} C_VEL
LIN {X 0,Y 594.331,Z 374.45,A -85,B 0,C 180,E1 -1062.094,E2 -1062.094} C_VEL
LIN {X 0,Y 594.342,Z 374.448,A -85,B 0,C 180,E1 -1064.218,E2 -1064.218} C_VEL
LIN {X 0,Y 594.365,Z 374.444,A -85,B 0,C 180,E1 -1066.321,E2 -1066.321} C_VEL
LIN {X 0,Y 594.335,Z 374.445,A -85,B 0,C 180,E1 -1068.956,E2 -1068.956} C_VEL
LIN {X 0,Y 594.377,Z 374.45,A -85,B 0,C 180,E1 -1071.843,E2 -1071.843} C_VEL
LIN {X 0,Y 594.357,Z 374.442,A -85,B 0,C 180,E1 -1074.572,E2 -1074.572} C_VEL
LIN {X 0,Y 594.377,Z 374.443,A -85,B 0,C 180,E1 -1077.289,E2 -1077.289} C_VEL
LIN {X 0,Y 594.414,Z 374.442,A -85,B 0,C 180,E1 -1080,E2 -1080} C_VEL
LIN {X 0,Y 594.367,Z 374.44,A -85,B 0,C 180,E1 -1082.711,E2 -1082.711} C_VEL
LIN {X 0,Y 594.365,Z 374.447,A -85,B 0,C 180,E1 -1085.428,E2 -1085.428} C_VEL
LIN {X 0,Y 594.376,Z 374.444,A -85,B 0,C 180,E1 -1088.157,E2 -1088.157} C_VEL
LIN {X 0,Y 594.335,Z 374.446,A -85,B 0,C 180,E1 -1091.044,E2 -1091.044} C_VEL
LIN {X 0,Y 594.368,Z 374.45,A -85,B 0,C 180,E1 -1093.679,E2 -1093.679} C_VEL
LIN {X 0,Y 594.329,Z 374.445,A -85,B 0,C 180,E1 -1096.696,E2 -1096.696} C_VEL
LIN {X 0,Y 594.335,Z 374.449,A -85,B 0,C 180,E1 -1099.336,E2 -1099.336} C_VEL
LIN {X 0,Y 594.344,Z 374.45,A -85,B 0,C 180,E1 -1101.504,E2 -1101.504} C_VEL
LIN {X 0,Y 594.348,Z 374.445,A -85,B 0,C 180,E1 -1104.448,E2 -1104.448} C_VEL
LIN {X 0,Y 594.337,Z 374.446,A -85,B 0,C 180,E1 -1106.702,E2 -1106.702} C_VEL
LIN {X 0,Y 594.357,Z 374.452,A -85,B 0,C 180,E1 -1109.777,E2 -1109.777} C_VEL
LIN {X 0,Y 594.344,Z 374.45,A -85,B 0,C 180,E1 -1112.149,E2 -1112.149} C_VEL
LIN {X 0,Y 594.347,Z 374.444,A -85,B 0,C 180,E1 -1114.582,E2 -1114.582} C_VEL
LIN {X 0,Y 594.353,Z 374.45,A -85,B 0,C 180,E1 -1117.603,E2 -1117.603} C_VEL
LIN {X 0,Y 594.326,Z 374.445,A -85,B 0,C 180,E1 -1120.571,E2 -1120.571} C_VEL
LIN {X 0,Y 594.315,Z 374.447,A -85,B 0,C 180,E1 -1122.846,E2 -1122.846} C_VEL
LIN {X 0,Y 594.357,Z 374.452,A -85,B 0,C 180,E1 -1125.761,E2 -1125.761} C_VEL
LIN {X 0,Y 594.354,Z 374.442,A -85,B 0,C 180,E1 -1128.533,E2 -1128.533} C_VEL
LIN {X 0,Y 594.328,Z 374.448,A -85,B 0,C 180,E1 -1131.303,E2 -1131.303} C_VEL
LIN {X 0,Y 594.34,Z 374.454,A -85,B 0,C 180,E1 -1133.754,E2 -1133.754} C_VEL
LIN {X 0,Y 594.343,Z 374.45,A -85,B 0,C 180,E1 -1136.236,E2 -1136.236} C_VEL
LIN {X 0,Y 594.313,Z 374.45,A -85,B 0,C 180,E1 -1138.646,E2 -1138.646} C_VEL
LIN {X 0,Y 594.333,Z 374.448,A -85,B 0,C 180,E1 -1141.051,E2 -1141.051} C_VEL
LIN {X 0,Y 594.364,Z 374.669,A -85,B 0,C 180,E1 -1143.386,E2 -1143.386} C_VEL
LIN {X 0,Y 595.226,Z 379.376,A -85,B 0,C 180,E1 -1143.971,E2 -1143.971} C_VEL
LIN {X 0,Y 595.024,Z 404.023,A -85,B 0,C 180,E1 -1146.691,E2 -1146.691} C_VEL
LIN {X 0,Y 594.831,Z 430.92,A -85,B 0,C 180,E1 -1149.601,E2 -1149.601} C_VEL
LIN {X 0,Y 594.657,Z 457.816,A -85,B 0,C 180,E1 -1152.46,E2 -1152.46} C_VEL
LIN {X 0,Y 594.542,Z 484.712,A -85,B 0,C 180,E1 -1155.277,E2 -1155.277} C_VEL
LIN {X 0,Y 594.557,Z 498.12,A -85,B 0,C 180,E1 -1156.641,E2 -1156.641} C_VEL
LIN {X 0,Y 594.756,Z 503.704,A -85,B 0,C 180,E1 -1156.721,E2 -1156.721} C_VEL
LIN {X 0,Y 594.665,Z 607.937,A -85,B 0,C 180,E1 -1157.999,E2 -1157.999} C_VEL
LIN {X 0,Y 594.635,Z 621.211,A -85,B 0,C 180,E1 -1158.301,E2 -1158.301} C_VEL
LIN {X 0,Y 594.596,Z 633.566,A -85,B 0,C 180,E1 -1158.718,E2 -1158.718} C_VEL
LIN {X 0,Y 594.537,Z 645.629,A -85,B 0,C 180,E1 -1159.27,E2 -1159.27} C_VEL
LIN {X 0,Y 594.473,Z 657.197,A -85,B 0,C 180,E1 -1159.957,E2 -1159.957} C_VEL
LIN {X 0,Y 594.414,Z 667.594,A -85,B 0,C 180,E1 -1160.729,E2 -1160.729} C_VEL
LIN {X 0,Y 594.383,Z 676.11,A -85,B 0,C 180,E1 -1161.5,E2 -1161.5} C_VEL
LIN {X 0,Y 594.347,Z 683.959,A -85,B 0,C 180,E1 -1162.355,E2 -1162.355} C_VEL
LIN {X 0,Y 594.283,Z 691.812,A -85,B 0,C 180,E1 -1163.408,E2 -1163.408} C_VEL
LIN {X 0,Y 594.289,Z 698.68,A -85,B 0,C 180,E1 -1164.571,E2 -1164.571} C_VEL
LIN {X 0,Y 594.27,Z 703.371,A -85,B 0,C 180,E1 -1165.591,E2 -1165.591} C_VEL
LIN {X 0,Y 594.267,Z 706.956,A -85,B 0,C 180,E1 -1166.61,E2 -1166.61} C_VEL
LIN {X 0,Y 594.226,Z 708.809,A -85,B 0,C 180,E1 -1167.288,E2 -1167.288} C_VEL
LIN {X 0,Y 594.241,Z 710.201,A -85,B 0,C 180,E1 -1167.967,E2 -1167.967} C_VEL
LIN {X 0,Y 594.239,Z 711.784,A -85,B 0,C 180,E1 -1169.322,E2 -1169.322} C_VEL
LIN {X 0,Y 594.236,Z 712,A -85,B 0,C 180,E1 -1170,E2 -1170} C_VEL
LIN {X 0,Y 594.247,Z 711.185,A -85,B 0,C 180,E1 -1171.355,E2 -1171.355} C_VEL
LIN {X 0,Y 594.241,Z 710.202,A -85,B 0,C 180,E1 -1172.033,E2 -1172.033} C_VEL
LIN {X 0,Y 594.226,Z 708.81,A -85,B 0,C 180,E1 -1172.712,E2 -1172.712} C_VEL
LIN {X 0,Y 594.289,Z 705.896,A -85,B 0,C 180,E1 -1173.729,E2 -1173.729} C_VEL
LIN {X 0,Y 594.241,Z 701.95,A -85,B 0,C 180,E1 -1174.749,E2 -1174.749} C_VEL
LIN {X 0,Y 594.304,Z 695.878,A -85,B 0,C 180,E1 -1175.939,E2 -1175.939} C_VEL
LIN {X 0,Y 594.308,Z 689.236,A -85,B 0,C 180,E1 -1176.962,E2 -1176.962} C_VEL
LIN {X 0,Y 594.359,Z 680.99,A -85,B 0,C 180,E1 -1177.986,E2 -1177.986} C_VEL
LIN {X 0,Y 594.382,Z 672.537,A -85,B 0,C 180,E1 -1178.842,E2 -1178.842} C_VEL
LIN {X 0,Y 594.431,Z 662.094,A -85,B 0,C 180,E1 -1179.699,E2 -1179.699} C_VEL
LIN {X 0,Y 594.493,Z 651.759,A -85,B 0,C 180,E1 -1180.386,E2 -1180.386} C_VEL
LIN {X 0,Y 594.562,Z 640.681,A -85,B 0,C 180,E1 -1180.975,E2 -1180.975} C_VEL
LIN {X 0,Y 594.6,Z 628.698,A -85,B 0,C 180,E1 -1181.464,E2 -1181.464} C_VEL
LIN {X 0,Y 594.648,Z 615.352,A -85,B 0,C 180,E1 -1181.85,E2 -1181.85} C_VEL
LIN {X 0,Y 594.695,Z 602.085,A -85,B 0,C 180,E1 -1182.087,E2 -1182.087} C_VEL
LIN {X 0,Y 594.608,Z 498.522,A -85,B 0,C 180,E1 -1183.347,E2 -1183.347} C_VEL
LIN {X 0,Y 594.484,Z 497.345,A -85,B 0,C 180,E1 -1183.415,E2 -1183.415} C_VEL
LIN {X 0,Y 594.619,Z 469.585,A -85,B 0,C 180,E1 -1186.303,E2 -1186.303} C_VEL
LIN {X 0,Y 594.742,Z 443.007,A -85,B 0,C 180,E1 -1189.109,E2 -1189.109} C_VEL
LIN {X 0,Y 594.922,Z 417.473,A -85,B 0,C 180,E1 -1191.846,E2 -1191.846} C_VEL
LIN {X 0,Y 595.158,Z 390.427,A -85,B 0,C 180,E1 -1194.801,E2 -1194.801} C_VEL
LIN {X 0,Y 595.212,Z 377.994,A -85,B 0,C 180,E1 -1196.185,E2 -1196.185} C_VEL
LIN {X 0,Y 594.359,Z 374.565,A -85,B 0,C 180,E1 -1196.641,E2 -1196.641} C_VEL
LIN {X 0,Y 594.348,Z 374.452,A -85,B 0,C 180,E1 -1199.778,E2 -1199.778} C_VEL
LIN {X 0,Y 594.334,Z 374.454,A -85,B 0,C 180,E1 -1202.149,E2 -1202.149} C_VEL
LIN {X 0,Y 594.341,Z 374.447,A -85,B 0,C 180,E1 -1204.583,E2 -1204.583} C_VEL
LIN {X 0,Y 594.352,Z 374.45,A -85,B 0,C 180,E1 -1207.603,E2 -1207.603} C_VEL
LIN {X 0,Y 594.326,Z 374.448,A -85,B 0,C 180,E1 -1210.571,E2 -1210.571} C_VEL
LIN {X 0,Y 594.319,Z 374.449,A -85,B 0,C 180,E1 -1212.847,E2 -1212.847} C_VEL
LIN {X 0,Y 594.339,Z 374.448,A -85,B 0,C 180,E1 -1215.194,E2 -1215.194} C_VEL
LIN {X 0,Y 594.376,Z 374.444,A -85,B 0,C 180,E1 -1218.153,E2 -1218.153} C_VEL
LIN {X 0,Y 594.361,Z 374.446,A -85,B 0,C 180,E1 -1221.193,E2 -1221.193} C_VEL
LIN {X 0,Y 594.348,Z 374.453,A -85,B 0,C 180,E1 -1223.755,E2 -1223.755} C_VEL
LIN {X 0,Y 594.364,Z 374.444,A -85,B 0,C 180,E1 -1226.238,E2 -1226.238} C_VEL
LIN {X 0,Y 594.363,Z 374.443,A -85,B 0,C 180,E1 -1228.649,E2 -1228.649} C_VEL
LIN {X 0,Y 594.38,Z 374.444,A -85,B 0,C 180,E1 -1231.043,E2 -1231.043} C_VEL
LIN {X 0,Y 594.363,Z 374.444,A -85,B 0,C 180,E1 -1234.055,E2 -1234.055} C_VEL
LIN {X 0,Y 594.377,Z 374.441,A -85,B 0,C 180,E1 -1236.295,E2 -1236.295} C_VEL
LIN {X 0,Y 594.405,Z 374.446,A -85,B 0,C 180,E1 -1239.224,E2 -1239.224} C_VEL
LIN {X 0,Y 594.352,Z 374.445,A -85,B 0,C 180,E1 -1242.095,E2 -1242.095} C_VEL
LIN {X 0,Y 594.361,Z 374.444,A -85,B 0,C 180,E1 -1244.219,E2 -1244.219} C_VEL
LIN {X 0,Y 594.431,Z 374.592,A -85,B 0,C 180,E1 -1246.91,E2 -1246.91} C_VEL
LIN {X 0,Y 594.628,Z 375.694,A -85,B 0,C 180,E1 -1247.023,E2 -1247.023} C_VEL
LIN {X 0,Y 594.686,Z 457.693,A -85,B 0,C 180,E1 -1248.043,E2 -1248.043} C_VEL
LIN {X 0,Y 594.648,Z 470.425,A -85,B 0,C 180,E1 -1248.323,E2 -1248.323} C_VEL
LIN {X 0,Y 594.594,Z 483.193,A -85,B 0,C 180,E1 -1248.748,E2 -1248.748} C_VEL
LIN {X 0,Y 594.564,Z 494.743,A -85,B 0,C 180,E1 -1249.271,E2 -1249.271} C_VEL
LIN {X 0,Y 594.463,Z 505.183,A -85,B 0,C 180,E1 -1249.871,E2 -1249.871} C_VEL
LIN {X 0,Y 594.419,Z 514.876,A -85,B 0,C 180,E1 -1250.558,E2 -1250.558} C_VEL
LIN {X 0,Y 594.378,Z 523.864,A -85,B 0,C 180,E1 -1251.329,E2 -1251.329} C_VEL
LIN {X 0,Y 594.347,Z 533.576,A -85,B 0,C 180,E1 -1252.355,E2 -1252.355} C_VEL
LIN {X 0,Y 594.305,Z 541.385,A -85,B 0,C 180,E1 -1253.39,E2 -1253.39} C_VEL
LIN {X 0,Y 594.303,Z 546.612,A -85,B 0,C 180,E1 -1254.231,E2 -1254.231} C_VEL
LIN {X 0,Y 594.24,Z 551.742,A -85,B 0,C 180,E1 -1255.251,E2 -1255.251} C_VEL
LIN {X 0,Y 594.288,Z 555.73,A -85,B 0,C 180,E1 -1256.271,E2 -1256.271} C_VEL
LIN {X 0,Y 594.225,Z 558.689,A -85,B 0,C 180,E1 -1257.288,E2 -1257.288} C_VEL
LIN {X 0,Y 594.241,Z 560.13,A -85,B 0,C 180,E1 -1257.967,E2 -1257.967} C_VEL
LIN {X 0,Y 594.24,Z 561.753,A -85,B 0,C 180,E1 -1259.322,E2 -1259.322} C_VEL
LIN {X 0,Y 594.236,Z 561.996,A -85,B 0,C 180,E1 -1260,E2 -1260} C_VEL
LIN {X 0,Y 594.248,Z 561.234,A -85,B 0,C 180,E1 -1261.355,E2 -1261.355} C_VEL
LIN {X 0,Y 594.242,Z 560.278,A -85,B 0,C 180,E1 -1262.033,E2 -1262.033} C_VEL
LIN {X 0,Y 594.226,Z 558.892,A -85,B 0,C 180,E1 -1262.712,E2 -1262.712} C_VEL
LIN {X 0,Y 594.289,Z 556.017,A -85,B 0,C 180,E1 -1263.729,E2 -1263.729} C_VEL
LIN {X 0,Y 594.241,Z 552.118,A -85,B 0,C 180,E1 -1264.749,E2 -1264.749} C_VEL
LIN {X 0,Y 594.299,Z 547.092,A -85,B 0,C 180,E1 -1265.769,E2 -1265.769} C_VEL
LIN {X 0,Y 594.308,Z 539.567,A -85,B 0,C 180,E1 -1266.962,E2 -1266.962} C_VEL
LIN {X 0,Y 594.36,Z 531.381,A -85,B 0,C 180,E1 -1267.986,E2 -1267.986} C_VEL
LIN {X 0,Y 594.368,Z 522.984,A -85,B 0,C 180,E1 -1268.842,E2 -1268.842} C_VEL
LIN {X 0,Y 594.432,Z 512.702,A -85,B 0,C 180,E1 -1269.699,E2 -1269.699} C_VEL
LIN {X 0,Y 594.516,Z 501.091,A -85,B 0,C 180,E1 -1270.472,E2 -1270.472} C_VEL
LIN {X 0,Y 594.571,Z 489.119,A -85,B 0,C 180,E1 -1271.089,E2 -1271.089} C_VEL
LIN {X 0,Y 594.599,Z 477.41,A -85,B 0,C 180,E1 -1271.55,E2 -1271.55} C_VEL
LIN {X 0,Y 594.641,Z 468.715,A -85,B 0,C 180,E1 -1271.812,E2 -1271.812} C_VEL
LIN {X 0,Y 594.075,Z 463.023,A -85,B 0,C 180,E1 -1271.961,E2 -1271.961} C_VEL
LIN {X 0,Y 591.267,Z 453.78,A -85,B 0,C 180,E1 -1272.179,E2 -1272.179} C_VEL
LIN {X 0,Y 588.431,Z 444.465,A -85,B 0,C 180,E1 -1272.359,E2 -1272.359} C_VEL
LIN {X 0,Y 587.782,Z 438.66,A -85,B 0,C 180,E1 -1272.441,E2 -1272.441} C_VEL
LIN {X 0,Y 587.665,Z 376.739,A -85,B 0,C 180,E1 -1273.208,E2 -1273.208} C_VEL
LIN {X 0,Y 587.39,Z 375.527,A -85,B 0,C 180,E1 -1273.316,E2 -1273.316} C_VEL
LIN {X 0,Y 587.323,Z 375.321,A -85,B 0,C 180,E1 -1275.975,E2 -1275.975} C_VEL
LIN {X 0,Y 587.35,Z 375.327,A -85,B 0,C 180,E1 -1278.849,E2 -1278.849} C_VEL
LIN {X 0,Y 587.322,Z 375.32,A -85,B 0,C 180,E1 -1281.774,E2 -1281.774} C_VEL
LIN {X 0,Y 587.35,Z 375.327,A -85,B 0,C 180,E1 -1284.759,E2 -1284.759} C_VEL
LIN {X 0,Y 587.318,Z 375.325,A -85,B 0,C 180,E1 -1287.047,E2 -1287.047} C_VEL
LIN {X 0,Y 587.349,Z 375.317,A -85,B 0,C 180,E1 -1289.38,E2 -1289.38} C_VEL
LIN {X 0,Y 587.345,Z 375.317,A -85,B 0,C 180,E1 -1291.835,E2 -1291.835} C_VEL
LIN {X 0,Y 587.346,Z 375.32,A -85,B 0,C 180,E1 -1294.347,E2 -1294.347} C_VEL
LIN {X 0,Y 587.344,Z 375.316,A -85,B 0,C 180,E1 -1297.608,E2 -1297.608} C_VEL
LIN {X 0,Y 587.312,Z 375.325,A -85,B 0,C 180,E1 -1300.255,E2 -1300.255} C_VEL
LIN {X 0,Y 587.306,Z 375.325,A -85,B 0,C 180,E1 -1303.117,E2 -1303.117} C_VEL
LIN {X 0,Y 587.316,Z 375.322,A -85,B 0,C 180,E1 -1306.049,E2 -1306.049} C_VEL
LIN {X 0,Y 587.335,Z 375.323,A -85,B 0,C 180,E1 -1308.925,E2 -1308.925} C_VEL
LIN {X 0,Y 587.32,Z 375.318,A -85,B 0,C 180,E1 -1311.52,E2 -1311.52} C_VEL
LIN {X 0,Y 587.29,Z 375.327,A -85,B 0,C 180,E1 -1314.1,E2 -1314.1} C_VEL
LIN {X 0,Y 587.336,Z 375.327,A -85,B 0,C 180,E1 -1316.603,E2 -1316.603} C_VEL
LIN {X 0,Y 587.323,Z 375.32,A -85,B 0,C 180,E1 -1319.493,E2 -1319.493} C_VEL
LIN {X 0,Y 587.305,Z 375.328,A -85,B 0,C 180,E1 -1322.18,E2 -1322.18} C_VEL
LIN {X 0,Y 587.357,Z 375.471,A -85,B 0,C 180,E1 -1323.722,E2 -1323.722} C_VEL
LIN {X 0,Y 588.337,Z 380.115,A -85,B 0,C 180,E1 -1324.34,E2 -1324.34} C_VEL
LIN {X 0,Y 588.114,Z 406.332,A -85,B 0,C 180,E1 -1327.384,E2 -1327.384} C_VEL
LIN {X 0,Y 587.881,Z 431.642,A -85,B 0,C 180,E1 -1330.262,E2 -1330.262} C_VEL
LIN {X 0,Y 587.649,Z 455.415,A -85,B 0,C 180,E1 -1332.919,E2 -1332.919} C_VEL
LIN {X 0,Y 587.532,Z 481.622,A -85,B 0,C 180,E1 -1335.812,E2 -1335.812} C_VEL
LIN {X 0,Y 587.513,Z 488.36,A -85,B 0,C 180,E1 -1336.522,E2 -1336.522} C_VEL
LIN {X 0,Y 587.879,Z 493.639,A -85,B 0,C 180,E1 -1336.607,E2 -1336.607} C_VEL
LIN {X 0,Y 587.743,Z 597.867,A -85,B 0,C 180,E1 -1337.899,E2 -1337.899} C_VEL
LIN {X 0,Y 587.711,Z 610.35,A -85,B 0,C 180,E1 -1338.183,E2 -1338.183} C_VEL
LIN {X 0,Y 587.629,Z 622.485,A -85,B 0,C 180,E1 -1338.586,E2 -1338.586} C_VEL
LIN {X 0,Y 587.555,Z 634.774,A -85,B 0,C 180,E1 -1339.141,E2 -1339.141} C_VEL
LIN {X 0,Y 587.475,Z 646.517,A -85,B 0,C 180,E1 -1339.837,E2 -1339.837} C_VEL
LIN {X 0,Y 587.365,Z 657.016,A -85,B 0,C 180,E1 -1340.617,E2 -1340.617} C_VEL
LIN {X 0,Y 587.31,Z 665.628,A -85,B 0,C 180,E1 -1341.397,E2 -1341.397} C_VEL
LIN {X 0,Y 587.272,Z 674.986,A -85,B 0,C 180,E1 -1342.436,E2 -1342.436} C_VEL
LIN {X 0,Y 587.247,Z 681.829,A -85,B 0,C 180,E1 -1343.376,E2 -1343.376} C_VEL
LIN {X 0,Y 587.211,Z 688.442,A -85,B 0,C 180,E1 -1344.506,E2 -1344.506} C_VEL
LIN {X 0,Y 587.188,Z 693.175,A -85,B 0,C 180,E1 -1345.538,E2 -1345.538} C_VEL
LIN {X 0,Y 587.193,Z 696.8,A -85,B 0,C 180,E1 -1346.569,E2 -1346.569} C_VEL
LIN {X 0,Y 587.131,Z 698.696,A -85,B 0,C 180,E1 -1347.256,E2 -1347.256} C_VEL
LIN {X 0,Y 587.14,Z 700.134,A -85,B 0,C 180,E1 -1347.942,E2 -1347.942} C_VEL
LIN {X 0,Y 587.14,Z 701.756,A -85,B 0,C 180,E1 -1349.314,E2 -1349.314} C_VEL
LIN {X 0,Y 587.137,Z 701.996,A -85,B 0,C 180,E1 -1350,E2 -1350} C_VEL
LIN {X 0,Y 587.14,Z 701.811,A -85,B 0,C 180,E1 -1350.686,E2 -1350.686} C_VEL
LIN {X 0,Y 587.141,Z 700.279,A -85,B 0,C 180,E1 -1352.058,E2 -1352.058} C_VEL
LIN {X 0,Y 587.132,Z 698.894,A -85,B 0,C 180,E1 -1352.744,E2 -1352.744} C_VEL
LIN {X 0,Y 587.213,Z 696.019,A -85,B 0,C 180,E1 -1353.774,E2 -1353.774} C_VEL
LIN {X 0,Y 587.147,Z 692.126,A -85,B 0,C 180,E1 -1354.806,E2 -1354.806} C_VEL
LIN {X 0,Y 587.229,Z 687.102,A -85,B 0,C 180,E1 -1355.839,E2 -1355.839} C_VEL
LIN {X 0,Y 587.245,Z 679.55,A -85,B 0,C 180,E1 -1357.046,E2 -1357.046} C_VEL
LIN {X 0,Y 587.287,Z 671.354,A -85,B 0,C 180,E1 -1358.083,E2 -1358.083} C_VEL
LIN {X 0,Y 587.338,Z 662.987,A -85,B 0,C 180,E1 -1358.949,E2 -1358.949} C_VEL
LIN {X 0,Y 587.419,Z 652.702,A -85,B 0,C 180,E1 -1359.816,E2 -1359.816} C_VEL
LIN {X 0,Y 587.517,Z 641.05,A -85,B 0,C 180,E1 -1360.598,E2 -1360.598} C_VEL
LIN {X 0,Y 587.596,Z 629.989,A -85,B 0,C 180,E1 -1361.182,E2 -1361.182} C_VEL
LIN {X 0,Y 587.63,Z 618.855,A -85,B 0,C 180,E1 -1361.641,E2 -1361.641} C_VEL
LIN {X 0,Y 587.695,Z 605.437,A -85,B 0,C 180,E1 -1362.036,E2 -1362.036} C_VEL
LIN {X 0,Y 587.769,Z 592.158,A -85,B 0,C 180,E1 -1362.276,E2 -1362.276} C_VEL
LIN {X 0,Y 587.753,Z 490.205,A -85,B 0,C 180,E1 -1363.528,E2 -1363.528} C_VEL
LIN {X 0,Y 587.503,Z 487.866,A -85,B 0,C 180,E1 -1363.6,E2 -1363.6} C_VEL
LIN {X 0,Y 587.641,Z 461.438,A -85,B 0,C 180,E1 -1366.502,E2 -1366.502} C_VEL
LIN {X 0,Y 587.844,Z 435.208,A -85,B 0,C 180,E1 -1369.427,E2 -1369.427} C_VEL
LIN {X 0,Y 588.079,Z 409.88,A -85,B 0,C 180,E1 -1372.299,E2 -1372.299} C_VEL
LIN {X 0,Y 588.332,Z 382.489,A -85,B 0,C 180,E1 -1375.471,E2 -1375.471} C_VEL
LIN {X 0,Y 588.237,Z 379.266,A -85,B 0,C 180,E1 -1375.855,E2 -1375.855} C_VEL
LIN {X 0,Y 587.337,Z 375.455,A -85,B 0,C 180,E1 -1376.375,E2 -1376.375} C_VEL
LIN {X 0,Y 587.317,Z 375.325,A -85,B 0,C 180,E1 -1379.381,E2 -1379.381} C_VEL
LIN {X 0,Y 587.317,Z 375.328,A -85,B 0,C 180,E1 -1381.831,E2 -1381.831} C_VEL
LIN {X 0,Y 587.337,Z 375.319,A -85,B 0,C 180,E1 -1384.346,E2 -1384.346} C_VEL
LIN {X 0,Y 587.32,Z 375.329,A -85,B 0,C 180,E1 -1387.61,E2 -1387.61} C_VEL
LIN {X 0,Y 587.306,Z 375.322,A -85,B 0,C 180,E1 -1390.255,E2 -1390.255} C_VEL
LIN {X 0,Y 587.286,Z 375.327,A -85,B 0,C 180,E1 -1393.115,E2 -1393.115} C_VEL
LIN {X 0,Y 587.302,Z 375.326,A -85,B 0,C 180,E1 -1396.047,E2 -1396.047} C_VEL
LIN {X 0,Y 587.307,Z 375.322,A -85,B 0,C 180,E1 -1398.84,E2 -1398.84} C_VEL
LIN {X 0,Y 587.315,Z 375.329,A -85,B 0,C 180,E1 -1401.519,E2 -1401.519} C_VEL
LIN {X 0,Y 587.279,Z 375.329,A -85,B 0,C 180,E1 -1404.099,E2 -1404.099} C_VEL
LIN {X 0,Y 587.337,Z 375.317,A -85,B 0,C 180,E1 -1406.889,E2 -1406.889} C_VEL
LIN {X 0,Y 587.325,Z 375.326,A -85,B 0,C 180,E1 -1409.493,E2 -1409.493} C_VEL
LIN {X 0,Y 587.302,Z 375.323,A -85,B 0,C 180,E1 -1412.317,E2 -1412.317} C_VEL
LIN {X 0,Y 587.311,Z 375.324,A -85,B 0,C 180,E1 -1415.239,E2 -1415.239} C_VEL
LIN {X 0,Y 587.308,Z 375.324,A -85,B 0,C 180,E1 -1418.225,E2 -1418.225} C_VEL
LIN {X 0,Y 587.33,Z 375.32,A -85,B 0,C 180,E1 -1421.15,E2 -1421.15} C_VEL
LIN {X 0,Y 587.298,Z 375.328,A -85,B 0,C 180,E1 -1424.024,E2 -1424.024} C_VEL
LIN {X 0,Y 587.35,Z 375.319,A -85,B 0,C 180,E1 -1426.154,E2 -1426.154} C_VEL
LIN {X 0,Y 587.295,Z 375.321,A -85,B 0,C 180,E1 -1428.961,E2 -1428.961} C_VEL
LIN {X 0,Y 587.336,Z 375.328,A -85,B 0,C 180,E1 -1431.744,E2 -1431.744} C_VEL
LIN {X 0,Y 587.327,Z 375.318,A -85,B 0,C 180,E1 -1434.507,E2 -1434.507} C_VEL
LIN {X 0,Y 587.344,Z 375.318,A -85,B 0,C 180,E1 -1437.257,E2 -1437.257} C_VEL
LIN {X 0,Y 587.383,Z 375.318,A -85,B 0,C 180,E1 -1440,E2 -1440} C_VEL
LIN {X 0,Y 587.336,Z 375.316,A -85,B 0,C 180,E1 -1442.743,E2 -1442.743} C_VEL
LIN {X 0,Y 587.333,Z 375.323,A -85,B 0,C 180,E1 -1445.493,E2 -1445.493} C_VEL
LIN {X 0,Y 587.332,Z 375.32,A -85,B 0,C 180,E1 -1448.256,E2 -1448.256} C_VEL
LIN {X 0,Y 587.301,Z 375.322,A -85,B 0,C 180,E1 -1451.107,E2 -1451.107} C_VEL
LIN {X 0,Y 587.345,Z 375.326,A -85,B 0,C 180,E1 -1453.846,E2 -1453.846} C_VEL
LIN {X 0,Y 587.282,Z 375.323,A -85,B 0,C 180,E1 -1456.791,E2 -1456.791} C_VEL
LIN {X 0,Y 587.287,Z 375.33,A -85,B 0,C 180,E1 -1459.577,E2 -1459.577} C_VEL
LIN {X 0,Y 587.306,Z 375.321,A -85,B 0,C 180,E1 -1462.515,E2 -1462.515} C_VEL
LIN {X 0,Y 587.304,Z 375.327,A -85,B 0,C 180,E1 -1465.518,E2 -1465.518} C_VEL
LIN {X 0,Y 587.287,Z 375.334,A -85,B 0,C 180,E1 -1467.821,E2 -1467.821} C_VEL
LIN {X 0,Y 587.318,Z 375.321,A -85,B 0,C 180,E1 -1470.506,E2 -1470.506} C_VEL
LIN {X 0,Y 587.287,Z 375.324,A -85,B 0,C 180,E1 -1473.103,E2 -1473.103} C_VEL
LIN {X 0,Y 587.262,Z 375.331,A -85,B 0,C 180,E1 -1475.532,E2 -1475.532} C_VEL
LIN {X 0,Y 587.306,Z 375.332,A -85,B 0,C 180,E1 -1477.834,E2 -1477.834} C_VEL
LIN {X 0,Y 587.285,Z 375.324,A -85,B 0,C 180,E1 -1480.257,E2 -1480.257} C_VEL
LIN {X 0,Y 587.278,Z 375.324,A -85,B 0,C 180,E1 -1483.114,E2 -1483.114} C_VEL
LIN {X 0,Y 587.301,Z 375.329,A -85,B 0,C 180,E1 -1486.047,E2 -1486.047} C_VEL
LIN {X 0,Y 587.282,Z 375.321,A -85,B 0,C 180,E1 -1488.931,E2 -1488.931} C_VEL
LIN {X 0,Y 587.285,Z 375.328,A -85,B 0,C 180,E1 -1491.517,E2 -1491.517} C_VEL
LIN {X 0,Y 587.27,Z 375.334,A -85,B 0,C 180,E1 -1494.098,E2 -1494.098} C_VEL
LIN {X 0,Y 587.305,Z 375.323,A -85,B 0,C 180,E1 -1496.601,E2 -1496.601} C_VEL
LIN {X 0,Y 587.31,Z 375.326,A -85,B 0,C 180,E1 -1499.495,E2 -1499.495} C_VEL
LIN {X 0,Y 587.286,Z 375.329,A -85,B 0,C 180,E1 -1502.32,E2 -1502.32} C_VEL
LIN {X 0,Y 587.327,Z 375.566,A -85,B 0,C 180,E1 -1503.146,E2 -1503.146} C_VEL
LIN {X 0,Y 588.463,Z 380.489,A -85,B 0,C 180,E1 -1503.775,E2 -1503.775} C_VEL
LIN {X 0,Y 588.211,Z 405.704,A -85,B 0,C 180,E1 -1506.592,E2 -1506.592} C_VEL
LIN {X 0,Y 587.957,Z 430.92,A -85,B 0,C 180,E1 -1509.352,E2 -1509.352} C_VEL
LIN {X 0,Y 587.719,Z 457.816,A -85,B 0,C 180,E1 -1512.246,E2 -1512.246} C_VEL
LIN {X 0,Y 587.563,Z 483.031,A -85,B 0,C 180,E1 -1514.92,E2 -1514.92} C_VEL
LIN {X 0,Y 587.499,Z 497.89,A -85,B 0,C 180,E1 -1516.466,E2 -1516.466} C_VEL
LIN {X 0,Y 587.902,Z 501.915,A -85,B 0,C 180,E1 -1516.542,E2 -1516.542} C_VEL
LIN {X 0,Y 587.744,Z 607.937,A -85,B 0,C 180,E1 -1517.855,E2 -1517.855} C_VEL
LIN {X 0,Y 587.682,Z 621.212,A -85,B 0,C 180,E1 -1518.16,E2 -1518.16} C_VEL
LIN {X 0,Y 587.628,Z 633.749,A -85,B 0,C 180,E1 -1518.59,E2 -1518.59} C_VEL
LIN {X 0,Y 587.561,Z 645.628,A -85,B 0,C 180,E1 -1519.141,E2 -1519.141} C_VEL
LIN {X 0,Y 587.455,Z 657.199,A -85,B 0,C 180,E1 -1519.836,E2 -1519.836} C_VEL
LIN {X 0,Y 587.393,Z 667.595,A -85,B 0,C 180,E1 -1520.618,E2 -1520.618} C_VEL
LIN {X 0,Y 587.322,Z 676.111,A -85,B 0,C 180,E1 -1521.397,E2 -1521.397} C_VEL
LIN {X 0,Y 587.274,Z 683.959,A -85,B 0,C 180,E1 -1522.263,E2 -1522.263} C_VEL
LIN {X 0,Y 587.23,Z 690.468,A -85,B 0,C 180,E1 -1523.126,E2 -1523.126} C_VEL
LIN {X 0,Y 587.236,Z 696.866,A -85,B 0,C 180,E1 -1524.161,E2 -1524.161} C_VEL
LIN {X 0,Y 587.147,Z 701.949,A -85,B 0,C 180,E1 -1525.194,E2 -1525.194} C_VEL
LIN {X 0,Y 587.213,Z 705.895,A -85,B 0,C 180,E1 -1526.226,E2 -1526.226} C_VEL
LIN {X 0,Y 587.132,Z 708.808,A -85,B 0,C 180,E1 -1527.256,E2 -1527.256} C_VEL
LIN {X 0,Y 587.14,Z 710.2,A -85,B 0,C 180,E1 -1527.942,E2 -1527.942} C_VEL
LIN {X 0,Y 587.14,Z 711.784,A -85,B 0,C 180,E1 -1529.314,E2 -1529.314} C_VEL
LIN {X 0,Y 587.137,Z 712,A -85,B 0,C 180,E1 -1530,E2 -1530} C_VEL
LIN {X 0,Y 587.147,Z 711.185,A -85,B 0,C 180,E1 -1531.372,E2 -1531.372} C_VEL
LIN {X 0,Y 587.14,Z 710.201,A -85,B 0,C 180,E1 -1532.058,E2 -1532.058} C_VEL
LIN {X 0,Y 587.132,Z 708.81,A -85,B 0,C 180,E1 -1532.744,E2 -1532.744} C_VEL
LIN {X 0,Y 587.213,Z 705.896,A -85,B 0,C 180,E1 -1533.774,E2 -1533.774} C_VEL
LIN {X 0,Y 587.147,Z 701.95,A -85,B 0,C 180,E1 -1534.806,E2 -1534.806} C_VEL
LIN {X 0,Y 587.217,Z 695.878,A -85,B 0,C 180,E1 -1536.011,E2 -1536.011} C_VEL
LIN {X 0,Y 587.245,Z 689.237,A -85,B 0,C 180,E1 -1537.046,E2 -1537.046} C_VEL
LIN {X 0,Y 587.3,Z 680.99,A -85,B 0,C 180,E1 -1538.083,E2 -1538.083} C_VEL
LIN {X 0,Y 587.343,Z 672.538,A -85,B 0,C 180,E1 -1538.949,E2 -1538.949} C_VEL
LIN {X 0,Y 587.419,Z 662.095,A -85,B 0,C 180,E1 -1539.816,E2 -1539.816} C_VEL
LIN {X 0,Y 587.513,Z 651.759,A -85,B 0,C 180,E1 -1540.511,E2 -1540.511} C_VEL
LIN {X 0,Y 587.584,Z 639.799,A -85,B 0,C 180,E1 -1541.149,E2 -1541.149} C_VEL
LIN {X 0,Y 587.639,Z 627.59,A -85,B 0,C 180,E1 -1541.639,E2 -1541.639} C_VEL
LIN {X 0,Y 587.704,Z 614.436,A -85,B 0,C 180,E1 -1542.014,E2 -1542.014} C_VEL
LIN {X 0,Y 587.779,Z 602.085,A -85,B 0,C 180,E1 -1542.231,E2 -1542.231} C_VEL
LIN {X 0,Y 587.814,Z 500.142,A -85,B 0,C 180,E1 -1543.482,E2 -1543.482} C_VEL
LIN {X 0,Y 587.494,Z 497.573,A -85,B 0,C 180,E1 -1543.556,E2 -1543.556} C_VEL
LIN {X 0,Y 587.684,Z 469.585,A -85,B 0,C 180,E1 -1546.5,E2 -1546.5} C_VEL
LIN {X 0,Y 587.822,Z 443.401,A -85,B 0,C 180,E1 -1549.3,E2 -1549.3} C_VEL
LIN {X 0,Y 588.061,Z 419.154,A -85,B 0,C 180,E1 -1551.93,E2 -1551.93} C_VEL
LIN {X 0,Y 588.326,Z 393.939,A -85,B 0,C 180,E1 -1554.715,E2 -1554.715} C_VEL
LIN {X 0,Y 588.462,Z 380.491,A -85,B 0,C 180,E1 -1556.225,E2 -1556.225} C_VEL
LIN {X 0,Y 587.304,Z 375.47,A -85,B 0,C 180,E1 -1556.879,E2 -1556.879} C_VEL
LIN {X 0,Y 587.294,Z 375.327,A -85,B 0,C 180,E1 -1559.383,E2 -1559.383} C_VEL
LIN {X 0,Y 587.295,Z 375.332,A -85,B 0,C 180,E1 -1561.827,E2 -1561.827} C_VEL
LIN {X 0,Y 587.317,Z 375.325,A -85,B 0,C 180,E1 -1564.343,E2 -1564.343} C_VEL
LIN {X 0,Y 587.307,Z 375.328,A -85,B 0,C 180,E1 -1567.611,E2 -1567.611} C_VEL
LIN {X 0,Y 587.288,Z 375.328,A -85,B 0,C 180,E1 -1570.257,E2 -1570.257} C_VEL
LIN {X 0,Y 587.281,Z 375.327,A -85,B 0,C 180,E1 -1573.114,E2 -1573.114} C_VEL
LIN {X 0,Y 587.3,Z 375.328,A -85,B 0,C 180,E1 -1576.047,E2 -1576.047} C_VEL
LIN {X 0,Y 587.306,Z 375.323,A -85,B 0,C 180,E1 -1578.929,E2 -1578.929} C_VEL
LIN {X 0,Y 587.315,Z 375.329,A -85,B 0,C 180,E1 -1581.519,E2 -1581.519} C_VEL
LIN {X 0,Y 587.281,Z 375.328,A -85,B 0,C 180,E1 -1584.099,E2 -1584.099} C_VEL
LIN {X 0,Y 587.328,Z 375.319,A -85,B 0,C 180,E1 -1586.603,E2 -1586.603} C_VEL
LIN {X 0,Y 587.335,Z 375.328,A -85,B 0,C 180,E1 -1589.491,E2 -1589.491} C_VEL
LIN {X 0,Y 587.306,Z 375.323,A -85,B 0,C 180,E1 -1592.18,E2 -1592.18} C_VEL
LIN {X 0,Y 587.348,Z 375.324,A -85,B 0,C 180,E1 -1595.241,E2 -1595.241} C_VEL
LIN {X 0,Y 587.32,Z 375.321,A -85,B 0,C 180,E1 -1598.226,E2 -1598.226} C_VEL
LIN {X 0,Y 587.35,Z 375.324,A -85,B 0,C 180,E1 -1601.151,E2 -1601.151} C_VEL
LIN {X 0,Y 587.321,Z 375.322,A -85,B 0,C 180,E1 -1604.025,E2 -1604.025} C_VEL
LIN {X 0,Y 587.363,Z 375.436,A -85,B 0,C 180,E1 -1606.749,E2 -1606.749} C_VEL
LIN {X 0,Y 587.563,Z 376.338,A -85,B 0,C 180,E1 -1606.864,E2 -1606.864} C_VEL
LIN {X 0,Y 587.844,Z 378.674,A -85,B 0,C 180,E1 -1606.914,E2 -1606.914} C_VEL
LIN {X 0,Y 587.743,Z 457.657,A -85,B 0,C 180,E1 -1607.899,E2 -1607.899} C_VEL
LIN {X 0,Y 587.693,Z 470.452,A -85,B 0,C 180,E1 -1608.183,E2 -1608.183} C_VEL
LIN {X 0,Y 587.628,Z 483.783,A -85,B 0,C 180,E1 -1608.635,E2 -1608.635} C_VEL
LIN {X 0,Y 587.586,Z 494.732,A -85,B 0,C 180,E1 -1609.142,E2 -1609.142} C_VEL
LIN {X 0,Y 587.454,Z 505.17,A -85,B 0,C 180,E1 -1609.749,E2 -1609.749} C_VEL
LIN {X 0,Y 587.393,Z 514.864,A -85,B 0,C 180,E1 -1610.444,E2 -1610.444} C_VEL
LIN {X 0,Y 587.336,Z 523.852,A -85,B 0,C 180,E1 -1611.224,E2 -1611.224} C_VEL
LIN {X 0,Y 587.274,Z 533.582,A -85,B 0,C 180,E1 -1612.263,E2 -1612.263} C_VEL
LIN {X 0,Y 587.247,Z 541.814,A -85,B 0,C 180,E1 -1613.376,E2 -1613.376} C_VEL
LIN {X 0,Y 587.211,Z 548.418,A -85,B 0,C 180,E1 -1614.506,E2 -1614.506} C_VEL
LIN {X 0,Y 587.188,Z 553.158,A -85,B 0,C 180,E1 -1615.538,E2 -1615.538} C_VEL
LIN {X 0,Y 587.193,Z 556.802,A -85,B 0,C 180,E1 -1616.569,E2 -1616.569} C_VEL
LIN {X 0,Y 587.131,Z 558.679,A -85,B 0,C 180,E1 -1617.256,E2 -1617.256} C_VEL
LIN {X 0,Y 587.14,Z 560.132,A -85,B 0,C 180,E1 -1617.942,E2 -1617.942} C_VEL
LIN {X 0,Y 587.14,Z 561.754,A -85,B 0,C 180,E1 -1619.314,E2 -1619.314} C_VEL
LIN {X 0,Y 587.137,Z 561.996,A -85,B 0,C 180,E1 -1620,E2 -1620} C_VEL
LIN {X 0,Y 587.148,Z 561.233,A -85,B 0,C 180,E1 -1621.372,E2 -1621.372} C_VEL
LIN {X 0,Y 587.141,Z 560.279,A -85,B 0,C 180,E1 -1622.058,E2 -1622.058} C_VEL
LIN {X 0,Y 587.193,Z 557.08,A -85,B 0,C 180,E1 -1623.431,E2 -1623.431} C_VEL
LIN {X 0,Y 587.189,Z 553.531,A -85,B 0,C 180,E1 -1624.462,E2 -1624.462} C_VEL
LIN {X 0,Y 587.211,Z 548.884,A -85,B 0,C 180,E1 -1625.494,E2 -1625.494} C_VEL
LIN {X 0,Y 587.212,Z 542.523,A -85,B 0,C 180,E1 -1626.604,E2 -1626.604} C_VEL
LIN {X 0,Y 587.272,Z 535.678,A -85,B 0,C 180,E1 -1627.564,E2 -1627.564} C_VEL
LIN {X 0,Y 587.305,Z 526.569,A -85,B 0,C 180,E1 -1628.603,E2 -1628.603} C_VEL
LIN {X 0,Y 587.393,Z 516.011,A -85,B 0,C 180,E1 -1629.556,E2 -1629.556} C_VEL
LIN {X 0,Y 587.448,Z 506.537,A -85,B 0,C 180,E1 -1630.251,E2 -1630.251} C_VEL
LIN {X 0,Y 587.537,Z 496.379,A -85,B 0,C 180,E1 -1630.859,E2 -1630.859} C_VEL
LIN {X 0,Y 587.605,Z 484.722,A -85,B 0,C 180,E1 -1631.414,E2 -1631.414} C_VEL
LIN {X 0,Y 587.704,Z 471.3,A -85,B 0,C 180,E1 -1631.883,E2 -1631.883} C_VEL
LIN {X 0,Y 587.735,Z 459.171,A -85,B 0,C 180,E1 -1632.167,E2 -1632.167} C_VEL
LIN {X 0,Y 587.782,Z 438.66,A -85,B 0,C 180,E1 -1632.441,E2 -1632.441} C_VEL
LIN {X 0,Y 587.152,Z 432.851,A -85,B 0,C 180,E1 -1632.526,E2 -1632.526} C_VEL
LIN {X 0,Y 581.563,Z 414.158,A -85,B 0,C 180,E1 -1632.879,E2 -1632.879} C_VEL
LIN {X 0,Y 580.93,Z 408.349,A -85,B 0,C 180,E1 -1632.966,E2 -1632.966} C_VEL
LIN {X 0,Y 580.794,Z 378.214,A -85,B 0,C 180,E1 -1633.345,E2 -1633.345} C_VEL
LIN {X 0,Y 580.409,Z 376.794,A -85,B 0,C 180,E1 -1633.412,E2 -1633.412} C_VEL
LIN {X 0,Y 580.309,Z 376.213,A -85,B 0,C 180,E1 -1633.571,E2 -1633.571} C_VEL
LIN {X 0,Y 580.277,Z 376.201,A -85,B 0,C 180,E1 -1636.175,E2 -1636.175} C_VEL
LIN {X 0,Y 580.3,Z 376.2,A -85,B 0,C 180,E1 -1639.151,E2 -1639.151} C_VEL
LIN {X 0,Y 580.273,Z 376.199,A -85,B 0,C 180,E1 -1642.053,E2 -1642.053} C_VEL
LIN {X 0,Y 580.304,Z 376.199,A -85,B 0,C 180,E1 -1645.08,E2 -1645.08} C_VEL
LIN {X 0,Y 580.285,Z 376.197,A -85,B 0,C 180,E1 -1648.186,E2 -1648.186} C_VEL
LIN {X 0,Y 580.286,Z 376.205,A -85,B 0,C 180,E1 -1650.694,E2 -1650.694} C_VEL
LIN {X 0,Y 580.286,Z 376.196,A -85,B 0,C 180,E1 -1653.313,E2 -1653.313} C_VEL
LIN {X 0,Y 580.248,Z 376.201,A -85,B 0,C 180,E1 -1655.756,E2 -1655.756} C_VEL
LIN {X 0,Y 580.29,Z 376.197,A -85,B 0,C 180,E1 -1658.146,E2 -1658.146} C_VEL
LIN {X 0,Y 580.297,Z 376.201,A -85,B 0,C 180,E1 -1660.844,E2 -1660.844} C_VEL
LIN {X 0,Y 580.244,Z 376.202,A -85,B 0,C 180,E1 -1663.661,E2 -1663.661} C_VEL
LIN {X 0,Y 580.269,Z 376.209,A -85,B 0,C 180,E1 -1666.61,E2 -1666.61} C_VEL
LIN {X 0,Y 580.297,Z 376.197,A -85,B 0,C 180,E1 -1669.156,E2 -1669.156} C_VEL
LIN {X 0,Y 580.288,Z 376.195,A -85,B 0,C 180,E1 -1671.928,E2 -1671.928} C_VEL
LIN {X 0,Y 580.25,Z 376.21,A -85,B 0,C 180,E1 -1674.452,E2 -1674.452} C_VEL
LIN {X 0,Y 580.29,Z 376.199,A -85,B 0,C 180,E1 -1676.975,E2 -1676.975} C_VEL
LIN {X 0,Y 580.284,Z 376.197,A -85,B 0,C 180,E1 -1679.424,E2 -1679.424} C_VEL
LIN {X 0,Y 580.259,Z 376.206,A -85,B 0,C 180,E1 -1682.149,E2 -1682.149} C_VEL
LIN {X 0,Y 580.3,Z 376.334,A -85,B 0,C 180,E1 -1683.535,E2 -1683.535} C_VEL
LIN {X 0,Y 581.512,Z 381.635,A -85,B 0,C 180,E1 -1684.209,E2 -1684.209} C_VEL
LIN {X 0,Y 581.303,Z 401.053,A -85,B 0,C 180,E1 -1686.486,E2 -1686.486} C_VEL
LIN {X 0,Y 581.062,Z 425.207,A -85,B 0,C 180,E1 -1689.281,E2 -1689.281} C_VEL
LIN {X 0,Y 580.785,Z 450.972,A -85,B 0,C 180,E1 -1692.209,E2 -1692.209} C_VEL
LIN {X 0,Y 580.551,Z 476.738,A -85,B 0,C 180,E1 -1695.093,E2 -1695.093} C_VEL
LIN {X 0,Y 580.511,Z 488.176,A -85,B 0,C 180,E1 -1696.345,E2 -1696.345} C_VEL
LIN {X 0,Y 580.972,Z 493.685,A -85,B 0,C 180,E1 -1696.445,E2 -1696.445} C_VEL
LIN {X 0,Y 580.823,Z 597.891,A -85,B 0,C 180,E1 -1697.753,E2 -1697.753} C_VEL
LIN {X 0,Y 580.767,Z 610.345,A -85,B 0,C 180,E1 -1698.04,E2 -1698.04} C_VEL
LIN {X 0,Y 580.675,Z 622.21,A -85,B 0,C 180,E1 -1698.437,E2 -1698.437} C_VEL
LIN {X 0,Y 580.561,Z 634.787,A -85,B 0,C 180,E1 -1699.009,E2 -1699.009} C_VEL
LIN {X 0,Y 580.454,Z 646.52,A -85,B 0,C 180,E1 -1699.712,E2 -1699.712} C_VEL
LIN {X 0,Y 580.345,Z 657.013,A -85,B 0,C 180,E1 -1700.503,E2 -1700.503} C_VEL
LIN {X 0,Y 580.268,Z 665.627,A -85,B 0,C 180,E1 -1701.292,E2 -1701.292} C_VEL
LIN {X 0,Y 580.221,Z 674.992,A -85,B 0,C 180,E1 -1702.343,E2 -1702.343} C_VEL
LIN {X 0,Y 580.17,Z 682.362,A -85,B 0,C 180,E1 -1703.377,E2 -1703.377} C_VEL
LIN {X 0,Y 580.139,Z 688.44,A -85,B 0,C 180,E1 -1704.439,E2 -1704.439} C_VEL
LIN {X 0,Y 580.108,Z 693.17,A -85,B 0,C 180,E1 -1705.483,E2 -1705.483} C_VEL
LIN {X 0,Y 580.123,Z 696.797,A -85,B 0,C 180,E1 -1706.527,E2 -1706.527} C_VEL
LIN {X 0,Y 580.043,Z 698.693,A -85,B 0,C 180,E1 -1707.222,E2 -1707.222} C_VEL
LIN {X 0,Y 580.039,Z 700.136,A -85,B 0,C 180,E1 -1707.917,E2 -1707.917} C_VEL
LIN {X 0,Y 580.04,Z 701.757,A -85,B 0,C 180,E1 -1709.306,E2 -1709.306} C_VEL
LIN {X 0,Y 580.038,Z 701.996,A -85,B 0,C 180,E1 -1710,E2 -1710} C_VEL
LIN {X 0,Y 580.047,Z 701.231,A -85,B 0,C 180,E1 -1711.389,E2 -1711.389} C_VEL
LIN {X 0,Y 580.04,Z 700.279,A -85,B 0,C 180,E1 -1712.083,E2 -1712.083} C_VEL
LIN {X 0,Y 580.044,Z 698.886,A -85,B 0,C 180,E1 -1712.778,E2 -1712.778} C_VEL
LIN {X 0,Y 580.11,Z 696.012,A -85,B 0,C 180,E1 -1713.821,E2 -1713.821} C_VEL
LIN {X 0,Y 580.053,Z 692.121,A -85,B 0,C 180,E1 -1714.865,E2 -1714.865} C_VEL
LIN {X 0,Y 580.16,Z 687.098,A -85,B 0,C 180,E1 -1715.91,E2 -1715.91} C_VEL
LIN {X 0,Y 580.158,Z 680.778,A -85,B 0,C 180,E1 -1716.958,E2 -1716.958} C_VEL
LIN {X 0,Y 580.231,Z 672.841,A -85,B 0,C 180,E1 -1718.007,E2 -1718.007} C_VEL
LIN {X 0,Y 580.298,Z 664.759,A -85,B 0,C 180,E1 -1718.883,E2 -1718.883} C_VEL
LIN {X 0,Y 580.367,Z 654.918,A -85,B 0,C 180,E1 -1719.761,E2 -1719.761} C_VEL
LIN {X 0,Y 580.503,Z 643.9,A -85,B 0,C 180,E1 -1720.551,E2 -1720.551} C_VEL
LIN {X 0,Y 580.57,Z 633.067,A -85,B 0,C 180,E1 -1721.168,E2 -1721.168} C_VEL
LIN {X 0,Y 580.696,Z 621.079,A -85,B 0,C 180,E1 -1721.696,E2 -1721.696} C_VEL
LIN {X 0,Y 580.749,Z 609.612,A -85,B 0,C 180,E1 -1722.072,E2 -1722.072} C_VEL
LIN {X 0,Y 580.825,Z 596.686,A -85,B 0,C 180,E1 -1722.358,E2 -1722.358} C_VEL
LIN {X 0,Y 580.836,Z 490.718,A -85,B 0,C 180,E1 -1723.685,E2 -1723.685} C_VEL
LIN {X 0,Y 580.511,Z 488.16,A -85,B 0,C 180,E1 -1723.745,E2 -1723.745} C_VEL
LIN {X 0,Y 580.686,Z 461.433,A -85,B 0,C 180,E1 -1726.705,E2 -1726.705} C_VEL
LIN {X 0,Y 580.927,Z 436.743,A -85,B 0,C 180,E1 -1729.492,E2 -1729.492} C_VEL
LIN {X 0,Y 581.222,Z 411.486,A -85,B 0,C 180,E1 -1732.389,E2 -1732.389} C_VEL
LIN {X 0,Y 581.547,Z 384.084,A -85,B 0,C 180,E1 -1735.597,E2 -1735.597} C_VEL
LIN {X 0,Y 581.45,Z 381.11,A -85,B 0,C 180,E1 -1735.943,E2 -1735.943} C_VEL
LIN {X 0,Y 580.288,Z 376.335,A -85,B 0,C 180,E1 -1736.557,E2 -1736.557} C_VEL
LIN {X 0,Y 580.279,Z 376.2,A -85,B 0,C 180,E1 -1739.305,E2 -1739.305} C_VEL
LIN {X 0,Y 580.287,Z 376.199,A -85,B 0,C 180,E1 -1742.202,E2 -1742.202} C_VEL
LIN {X 0,Y 580.279,Z 376.198,A -85,B 0,C 180,E1 -1744.697,E2 -1744.697} C_VEL
LIN {X 0,Y 580.274,Z 376.201,A -85,B 0,C 180,E1 -1747.271,E2 -1747.271} C_VEL
LIN {X 0,Y 580.286,Z 376.196,A -85,B 0,C 180,E1 -1750.269,E2 -1750.269} C_VEL
LIN {X 0,Y 580.251,Z 376.201,A -85,B 0,C 180,E1 -1752.709,E2 -1752.709} C_VEL
LIN {X 0,Y 580.254,Z 376.207,A -85,B 0,C 180,E1 -1755.611,E2 -1755.611} C_VEL
LIN {X 0,Y 580.252,Z 376.203,A -85,B 0,C 180,E1 -1758.228,E2 -1758.228} C_VEL
LIN {X 0,Y 580.265,Z 376.2,A -85,B 0,C 180,E1 -1760.964,E2 -1760.964} C_VEL
LIN {X 0,Y 580.242,Z 376.21,A -85,B 0,C 180,E1 -1763.594,E2 -1763.594} C_VEL
LIN {X 0,Y 580.279,Z 376.199,A -85,B 0,C 180,E1 -1766.143,E2 -1766.143} C_VEL
LIN {X 0,Y 580.269,Z 376.198,A -85,B 0,C 180,E1 -1768.614,E2 -1768.614} C_VEL
LIN {X 0,Y 580.253,Z 376.2,A -85,B 0,C 180,E1 -1771.022,E2 -1771.022} C_VEL
LIN {X 0,Y 580.259,Z 376.21,A -85,B 0,C 180,E1 -1773.674,E2 -1773.674} C_VEL
LIN {X 0,Y 580.267,Z 376.198,A -85,B 0,C 180,E1 -1776.441,E2 -1776.441} C_VEL
LIN {X 0,Y 580.261,Z 376.205,A -85,B 0,C 180,E1 -1779.437,E2 -1779.437} C_VEL
LIN {X 0,Y 580.245,Z 376.21,A -85,B 0,C 180,E1 -1781.644,E2 -1781.644} C_VEL
LIN {X 0,Y 580.271,Z 376.198,A -85,B 0,C 180,E1 -1784.546,E2 -1784.546} C_VEL
LIN {X 0,Y 580.253,Z 376.2,A -85,B 0,C 180,E1 -1786.695,E2 -1786.695} C_VEL
LIN {X 0,Y 580.272,Z 376.195,A -85,B 0,C 180,E1 -1788.826,E2 -1788.826} C_VEL
LIN {X 0,Y 580.304,Z 376.202,A -85,B 0,C 180,E1 -1791.644,E2 -1791.644} C_VEL
LIN {X 0,Y 580.296,Z 376.194,A -85,B 0,C 180,E1 -1794.44,E2 -1794.44} C_VEL
LIN {X 0,Y 580.311,Z 376.194,A -85,B 0,C 180,E1 -1797.223,E2 -1797.223} C_VEL
LIN {X 0,Y 580.351,Z 376.194,A -85,B 0,C 180,E1 -1800,E2 -1800} C_VEL
LIN {X 0,Y 580.304,Z 376.191,A -85,B 0,C 180,E1 -1802.777,E2 -1802.777} C_VEL
LIN {X 0,Y 580.302,Z 376.2,A -85,B 0,C 180,E1 -1805.56,E2 -1805.56} C_VEL
LIN {X 0,Y 580.298,Z 376.195,A -85,B 0,C 180,E1 -1808.357,E2 -1808.357} C_VEL
LIN {X 0,Y 580.272,Z 376.198,A -85,B 0,C 180,E1 -1811.174,E2 -1811.174} C_VEL
LIN {X 0,Y 580.305,Z 376.2,A -85,B 0,C 180,E1 -1814.017,E2 -1814.017} C_VEL
LIN {X 0,Y 580.231,Z 376.201,A -85,B 0,C 180,E1 -1816.9,E2 -1816.9} C_VEL
LIN {X 0,Y 580.266,Z 376.209,A -85,B 0,C 180,E1 -1819.824,E2 -1819.824} C_VEL
LIN {X 0,Y 580.279,Z 376.195,A -85,B 0,C 180,E1 -1822.803,E2 -1822.803} C_VEL
LIN {X 0,Y 580.251,Z 376.211,A -85,B 0,C 180,E1 -1825.851,E2 -1825.851} C_VEL
LIN {X 0,Y 580.225,Z 376.206,A -85,B 0,C 180,E1 -1828.19,E2 -1828.19} C_VEL
LIN {X 0,Y 580.268,Z 376.198,A -85,B 0,C 180,E1 -1830.691,E2 -1830.691} C_VEL
LIN {X 0,Y 580.271,Z 376.2,A -85,B 0,C 180,E1 -1833.311,E2 -1833.311} C_VEL
LIN {X 0,Y 580.221,Z 376.212,A -85,B 0,C 180,E1 -1835.752,E2 -1835.752} C_VEL
LIN {X 0,Y 580.268,Z 376.203,A -85,B 0,C 180,E1 -1838.148,E2 -1838.148} C_VEL
LIN {X 0,Y 580.237,Z 376.197,A -85,B 0,C 180,E1 -1840.849,E2 -1840.849} C_VEL
LIN {X 0,Y 580.226,Z 376.208,A -85,B 0,C 180,E1 -1843.663,E2 -1843.663} C_VEL
LIN {X 0,Y 580.235,Z 376.205,A -85,B 0,C 180,E1 -1846.337,E2 -1846.337} C_VEL
LIN {X 0,Y 580.236,Z 376.198,A -85,B 0,C 180,E1 -1849.151,E2 -1849.151} C_VEL
LIN {X 0,Y 580.27,Z 376.208,A -85,B 0,C 180,E1 -1851.93,E2 -1851.93} C_VEL
LIN {X 0,Y 580.214,Z 376.208,A -85,B 0,C 180,E1 -1854.45,E2 -1854.45} C_VEL
LIN {X 0,Y 580.24,Z 376.203,A -85,B 0,C 180,E1 -1856.972,E2 -1856.972} C_VEL
LIN {X 0,Y 580.268,Z 376.203,A -85,B 0,C 180,E1 -1859.423,E2 -1859.423} C_VEL
LIN {X 0,Y 580.233,Z 376.207,A -85,B 0,C 180,E1 -1862.154,E2 -1862.154} C_VEL
LIN {X 0,Y 580.265,Z 376.339,A -85,B 0,C 180,E1 -1862.938,E2 -1862.938} C_VEL
LIN {X 0,Y 581.608,Z 381.912,A -85,B 0,C 180,E1 -1863.631,E2 -1863.631} C_VEL
LIN {X 0,Y 581.445,Z 402.342,A -85,B 0,C 180,E1 -1865.924,E2 -1865.924} C_VEL
LIN {X 0,Y 581.148,Z 427.558,A -85,B 0,C 180,E1 -1868.728,E2 -1868.728} C_VEL
LIN {X 0,Y 580.864,Z 454.454,A -85,B 0,C 180,E1 -1871.664,E2 -1871.664} C_VEL
LIN {X 0,Y 580.61,Z 479.669,A -85,B 0,C 180,E1 -1874.376,E2 -1874.376} C_VEL
LIN {X 0,Y 580.516,Z 497.886,A -85,B 0,C 180,E1 -1876.3,E2 -1876.3} C_VEL
LIN {X 0,Y 580.979,Z 503.704,A -85,B 0,C 180,E1 -1876.4,E2 -1876.4} C_VEL
LIN {X 0,Y 580.819,Z 607.937,A -85,B 0,C 180,E1 -1877.708,E2 -1877.708} C_VEL
LIN {X 0,Y 580.736,Z 621.213,A -85,B 0,C 180,E1 -1878.017,E2 -1878.017} C_VEL
LIN {X 0,Y 580.678,Z 634.489,A -85,B 0,C 180,E1 -1878.481,E2 -1878.481} C_VEL
LIN {X 0,Y 580.564,Z 645.627,A -85,B 0,C 180,E1 -1879.008,E2 -1879.008} C_VEL
LIN {X 0,Y 580.429,Z 657.2,A -85,B 0,C 180,E1 -1879.712,E2 -1879.712} C_VEL
LIN {X 0,Y 580.344,Z 667.597,A -85,B 0,C 180,E1 -1880.503,E2 -1880.503} C_VEL
LIN {X 0,Y 580.271,Z 676.111,A -85,B 0,C 180,E1 -1881.292,E2 -1881.292} C_VEL
LIN {X 0,Y 580.222,Z 683.959,A -85,B 0,C 180,E1 -1882.168,E2 -1882.168} C_VEL
LIN {X 0,Y 580.154,Z 691.649,A -85,B 0,C 180,E1 -1883.221,E2 -1883.221} C_VEL
LIN {X 0,Y 580.139,Z 698.679,A -85,B 0,C 180,E1 -1884.438,E2 -1884.438} C_VEL
LIN {X 0,Y 580.108,Z 703.371,A -85,B 0,C 180,E1 -1885.483,E2 -1885.483} C_VEL
LIN {X 0,Y 580.123,Z 706.956,A -85,B 0,C 180,E1 -1886.527,E2 -1886.527} C_VEL
LIN {X 0,Y 580.043,Z 708.808,A -85,B 0,C 180,E1 -1887.222,E2 -1887.222} C_VEL
LIN {X 0,Y 580.039,Z 710.199,A -85,B 0,C 180,E1 -1887.917,E2 -1887.917} C_VEL
LIN {X 0,Y 580.04,Z 711.784,A -85,B 0,C 180,E1 -1889.306,E2 -1889.306} C_VEL
LIN {X 0,Y 580.037,Z 712,A -85,B 0,C 180,E1 -1890,E2 -1890} C_VEL
LIN {X 0,Y 580.046,Z 711.186,A -85,B 0,C 180,E1 -1891.388,E2 -1891.388} C_VEL
LIN {X 0,Y 580.039,Z 710.201,A -85,B 0,C 180,E1 -1892.083,E2 -1892.083} C_VEL
LIN {X 0,Y 580.043,Z 708.81,A -85,B 0,C 180,E1 -1892.778,E2 -1892.778} C_VEL
LIN {X 0,Y 580.11,Z 705.896,A -85,B 0,C 180,E1 -1893.821,E2 -1893.821} C_VEL
LIN {X 0,Y 580.053,Z 701.949,A -85,B 0,C 180,E1 -1894.865,E2 -1894.865} C_VEL
LIN {X 0,Y 580.139,Z 695.877,A -85,B 0,C 180,E1 -1896.085,E2 -1896.085} C_VEL
LIN {X 0,Y 580.184,Z 689.237,A -85,B 0,C 180,E1 -1897.132,E2 -1897.132} C_VEL
LIN {X 0,Y 580.25,Z 680.99,A -85,B 0,C 180,E1 -1898.182,E2 -1898.182} C_VEL
LIN {X 0,Y 580.308,Z 672.538,A -85,B 0,C 180,E1 -1899.058,E2 -1899.058} C_VEL
LIN {X 0,Y 580.42,Z 662.097,A -85,B 0,C 180,E1 -1899.936,E2 -1899.936} C_VEL
LIN {X 0,Y 580.517,Z 651.757,A -85,B 0,C 180,E1 -1900.639,E2 -1900.639} C_VEL
LIN {X 0,Y 580.598,Z 640.231,A -85,B 0,C 180,E1 -1901.265,E2 -1901.265} C_VEL
LIN {X 0,Y 580.682,Z 627.472,A -85,B 0,C 180,E1 -1901.785,E2 -1901.785} C_VEL
LIN {X 0,Y 580.759,Z 614.435,A -85,B 0,C 180,E1 -1902.16,E2 -1902.16} C_VEL
LIN {X 0,Y 580.863,Z 602.085,A -85,B 0,C 180,E1 -1902.379,E2 -1902.379} C_VEL
LIN {X 0,Y 580.795,Z 500.142,A -85,B 0,C 180,E1 -1903.648,E2 -1903.648} C_VEL
LIN {X 0,Y 580.516,Z 497.575,A -85,B 0,C 180,E1 -1903.722,E2 -1903.722} C_VEL
LIN {X 0,Y 580.73,Z 469.585,A -85,B 0,C 180,E1 -1906.704,E2 -1906.704} C_VEL
LIN {X 0,Y 580.932,Z 443.797,A -85,B 0,C 180,E1 -1909.495,E2 -1909.495} C_VEL
LIN {X 0,Y 581.266,Z 417.473,A -85,B 0,C 180,E1 -1912.387,E2 -1912.387} C_VEL
LIN {X 0,Y 581.592,Z 392.258,A -85,B 0,C 180,E1 -1915.212,E2 -1915.212} C_VEL
LIN {X 0,Y 581.573,Z 381.799,A -85,B 0,C 180,E1 -1916.372,E2 -1916.372} C_VEL
LIN {X 0,Y 580.262,Z 376.317,A -85,B 0,C 180,E1 -1917.037,E2 -1917.037} C_VEL
LIN {X 0,Y 580.255,Z 376.209,A -85,B 0,C 180,E1 -1919.775,E2 -1919.775} C_VEL
LIN {X 0,Y 580.269,Z 376.206,A -85,B 0,C 180,E1 -1922.203,E2 -1922.203} C_VEL
LIN {X 0,Y 580.265,Z 376.201,A -85,B 0,C 180,E1 -1924.698,E2 -1924.698} C_VEL
LIN {X 0,Y 580.263,Z 376.202,A -85,B 0,C 180,E1 -1927.271,E2 -1927.271} C_VEL
LIN {X 0,Y 580.251,Z 376.205,A -85,B 0,C 180,E1 -1930.265,E2 -1930.265} C_VEL
LIN {X 0,Y 580.247,Z 376.202,A -85,B 0,C 180,E1 -1932.709,E2 -1932.709} C_VEL
LIN {X 0,Y 580.252,Z 376.209,A -85,B 0,C 180,E1 -1935.611,E2 -1935.611} C_VEL
LIN {X 0,Y 580.25,Z 376.204,A -85,B 0,C 180,E1 -1938.228,E2 -1938.228} C_VEL
LIN {X 0,Y 580.265,Z 376.2,A -85,B 0,C 180,E1 -1940.964,E2 -1940.964} C_VEL
LIN {X 0,Y 580.243,Z 376.212,A -85,B 0,C 180,E1 -1943.594,E2 -1943.594} C_VEL
LIN {X 0,Y 580.308,Z 376.196,A -85,B 0,C 180,E1 -1946.145,E2 -1946.145} C_VEL
LIN {X 0,Y 580.274,Z 376.198,A -85,B 0,C 180,E1 -1948.614,E2 -1948.614} C_VEL
LIN {X 0,Y 580.29,Z 376.199,A -85,B 0,C 180,E1 -1951.024,E2 -1951.024} C_VEL
LIN {X 0,Y 580.26,Z 376.201,A -85,B 0,C 180,E1 -1954.149,E2 -1954.149} C_VEL
LIN {X 0,Y 580.274,Z 376.199,A -85,B 0,C 180,E1 -1956.442,E2 -1956.442} C_VEL
LIN {X 0,Y 580.276,Z 376.207,A -85,B 0,C 180,E1 -1959.437,E2 -1959.437} C_VEL
LIN {X 0,Y 580.267,Z 376.205,A -85,B 0,C 180,E1 -1961.645,E2 -1961.645} C_VEL
LIN {X 0,Y 580.278,Z 376.202,A -85,B 0,C 180,E1 -1963.825,E2 -1963.825} C_VEL
LIN {X 0,Y 580.326,Z 376.355,A -85,B 0,C 180,E1 -1966.608,E2 -1966.608} C_VEL
LIN {X 0,Y 580.51,Z 377.232,A -85,B 0,C 180,E1 -1966.713,E2 -1966.713} C_VEL
LIN {X 0,Y 580.95,Z 378.72,A -85,B 0,C 180,E1 -1966.756,E2 -1966.756} C_VEL
LIN {X 0,Y 580.827,Z 457.621,A -85,B 0,C 180,E1 -1967.753,E2 -1967.753} C_VEL
LIN {X 0,Y 580.737,Z 469.59,A -85,B 0,C 180,E1 -1968.017,E2 -1968.017} C_VEL
LIN {X 0,Y 580.67,Z 483.39,A -85,B 0,C 180,E1 -1968.481,E2 -1968.481} C_VEL
LIN {X 0,Y 580.597,Z 494.721,A -85,B 0,C 180,E1 -1969.009,E2 -1969.009} C_VEL
LIN {X 0,Y 580.462,Z 505.157,A -85,B 0,C 180,E1 -1969.624,E2 -1969.624} C_VEL
LIN {X 0,Y 580.374,Z 514.852,A -85,B 0,C 180,E1 -1970.327,E2 -1970.327} C_VEL
LIN {X 0,Y 580.305,Z 523.841,A -85,B 0,C 180,E1 -1971.117,E2 -1971.117} C_VEL
LIN {X 0,Y 580.242,Z 532.097,A -85,B 0,C 180,E1 -1971.993,E2 -1971.993} C_VEL
LIN {X 0,Y 580.159,Z 540.163,A -85,B 0,C 180,E1 -1973.042,E2 -1973.042} C_VEL
LIN {X 0,Y 580.165,Z 546.609,A -85,B 0,C 180,E1 -1974.09,E2 -1974.09} C_VEL
LIN {X 0,Y 580.052,Z 551.729,A -85,B 0,C 180,E1 -1975.135,E2 -1975.135} C_VEL
LIN {X 0,Y 580.109,Z 555.714,A -85,B 0,C 180,E1 -1976.179,E2 -1976.179} C_VEL
LIN {X 0,Y 580.043,Z 558.669,A -85,B 0,C 180,E1 -1977.222,E2 -1977.222} C_VEL
LIN {X 0,Y 580.039,Z 560.133,A -85,B 0,C 180,E1 -1977.917,E2 -1977.917} C_VEL
LIN {X 0,Y 580.04,Z 561.746,A -85,B 0,C 180,E1 -1979.306,E2 -1979.306} C_VEL
LIN {X 0,Y 580.038,Z 561.996,A -85,B 0,C 180,E1 -1980,E2 -1980} C_VEL
LIN {X 0,Y 580.047,Z 561.231,A -85,B 0,C 180,E1 -1981.389,E2 -1981.389} C_VEL
